SPLINE
SPL {X  -145.877, Y  +737.201, Z    +0.000, E1   +34.468, E3 -287162.055}
SPL {X  -152.550, Y  +719.721, Z    +0.000, E1   +27.728, E3 -287177.544}
SPL {X  -157.145, Y  +701.536, Z    +0.000, E1   +19.368, E3 -287186.999}
SPL {X  -159.035, Y  +688.952, Z    +0.000, E1   +12.676, E3 -287191.040}
SPL {X  -159.756, Y  +680.154, Z    +0.000, E1    +7.520, E3 -287192.766}
SPL {X  -159.986, Y  +672.560, Z    +0.000, E1    +2.636, E3 -287193.664}
SPL {X  -159.990, Y  +668.344, Z    +0.000, E1    -0.618, E3 -287193.931}
SPL {X  -159.990, Y  +664.070, Z    +0.000, E1    -5.025, E3 -287194.259}
SPL {X  -159.990, Y  +656.953, Z    +0.000, E1   -13.960, E3 -287195.325}
SPL {X  -159.990, Y  +644.589, Z    +0.000, E1   -29.011, E3 -287198.737}
SPL {X  -159.990, Y  +605.095, Z    +0.000, E1   -49.514, E3 -287223.828}
SPL {X  -159.990, Y  +543.998, Z    +0.000, E1   -54.483, E3 -287289.818}
SPL {X  -159.990, Y  +535.878, Z    +0.000, E1   -54.465, E3 -287302.152}
SPL {X  -159.990, Y  +529.394, Z    +0.000, E1   -54.464, E3 -287311.982}
SPL {X  -159.990, Y  +521.536, Z    +0.000, E1   -54.480, E3 -287323.864}
SPL {X  -159.990, Y  +512.119, Z    +0.000, E1   -54.487, E3 -287338.110}
SPL {X  -159.990, Y  +504.581, Z    +0.000, E1   -54.460, E3 -287349.569}
SPL {X  -159.990, Y  +497.571, Z    +0.000, E1   -54.478, E3 -287360.155}
SPL {X  -159.990, Y  +490.343, Z    +0.000, E1   -54.468, E3 -287371.121}
SPL {X  -159.990, Y  +483.191, Z    +0.000, E1   -54.478, E3 -287381.937}
SPL {X  -159.990, Y  +475.502, Z    +0.000, E1   -54.476, E3 -287393.586}
SPL {X  -159.990, Y  +448.520, Z    +0.000, E1   -58.543, E3 -287405.215}
SPL {X  -159.990, Y  +438.044, Z    +0.000, E1   -58.687, E3 -287417.852}
SPL {X  -159.990, Y  +431.936, Z    +0.000, E1   -57.955, E3 -287430.671}
SPL {X  -159.990, Y  +427.293, Z    +0.000, E1   -56.830, E3 -287444.377}
SPL {X  -159.990, Y  +423.841, Z    +0.000, E1   -55.679, E3 -287456.479}
SPL {X  -159.990, Y  +418.232, Z    +0.000, E1   -55.048, E3 -287468.833}
SPL {X  -159.990, Y  +410.722, Z    +0.000, E1   -54.900, E3 -287480.816}
SPL {X  -159.990, Y  +402.790, Z    +0.000, E1   -54.930, E3 -287492.591}
SPL {X  -159.990, Y  +392.953, Z    +0.000, E1   -54.918, E3 -287507.285}
SPL {X  -159.990, Y  +383.354, Z    +0.000, E1   -54.920, E3 -287521.595}
SPL {X  -159.769, Y  +374.091, Z    +0.000, E1   -54.882, E3 -287535.627}
SPL {X  -158.996, Y  +364.689, Z    +0.000, E1   -54.773, E3 -287550.424}
SPL {X  -157.966, Y  +357.131, Z    +0.000, E1   -54.559, E3 -287562.831}
SPL {X  -156.775, Y  +350.586, Z    +0.000, E1   -54.373, E3 -287573.805}
SPL {X  -155.027, Y  +342.959, Z    +0.000, E1   -54.074, E3 -287586.978}
SPL {X  -152.882, Y  +335.340, Z    +0.000, E1   -53.695, E3 -287600.520}
SPL {X  -151.019, Y  +329.680, Z    +0.000, E1   -53.334, E3 -287610.877}
SPL {X  -148.682, Y  +323.421, Z    +0.000, E1   -52.939, E3 -287622.480}
SPL {X  -145.914, Y  +316.881, Z    +0.000, E1   -52.402, E3 -287634.944}
SPL {X  -142.795, Y  +310.344, Z    +0.000, E1   -51.829, E3 -287647.600}
SPL {X  -132.354, Y  +292.616, Z    +0.000, E1   -44.164, E3 -287746.012}
ENDSPLINE

SPLINE
SPL {X  -150.910, Y  +329.369, Z    +0.000, E1   -29.678, E3 -287818.407}
SPL {X  -156.829, Y  +350.854, Z    +0.000, E1   -20.141, E3 -287830.960}
SPL {X  -159.049, Y  +365.169, Z    +0.000, E1   -12.580, E3 -287835.704}
SPL {X  -159.776, Y  +374.231, Z    +0.000, E1    -7.281, E3 -287837.590}
SPL {X  -159.986, Y  +381.380, Z    +0.000, E1    -2.685, E3 -287838.436}
SPL {X  -159.990, Y  +384.493, Z    +0.000, E1    -0.324, E3 -287838.644}
SPL {X  -159.990, Y  +387.327, Z    +0.000, E1    +2.137, E3 -287838.827}
SPL {X  -159.990, Y  +392.053, Z    +0.000, E1    +7.477, E3 -287839.292}
SPL {X  -159.990, Y  +396.158, Z    +0.000, E1   +12.775, E3 -287839.918}
SPL {X  -159.990, Y  +401.377, Z    +0.000, E1   +19.398, E3 -287841.098}
SPL {X  -159.990, Y  +411.365, Z    +0.000, E1   +30.630, E3 -287844.306}
SPL {X  -159.990, Y  +450.467, Z    +0.000, E1   +50.183, E3 -287867.955}
SPL {X  -159.990, Y  +509.934, Z    +0.000, E1   +54.923, E3 -287930.574}
SPL {X  -159.990, Y  +516.848, Z    +0.000, E1   +54.930, E3 -287940.862}
SPL {X  -159.990, Y  +524.818, Z    +0.000, E1   +54.933, E3 -287952.734}
SPL {X  -159.990, Y  +532.100, Z    +0.000, E1   +54.924, E3 -287963.587}
SPL {X  -159.990, Y  +539.391, Z    +0.000, E1   +54.933, E3 -287974.439}
SPL {X  -159.990, Y  +546.283, Z    +0.000, E1   +54.924, E3 -287984.711}
SPL {X  -159.990, Y  +553.734, Z    +0.000, E1   +54.938, E3 -287995.797}
SPL {X  -159.990, Y  +560.983, Z    +0.000, E1   +54.918, E3 -288006.635}
SPL {X  -159.990, Y  +567.462, Z    +0.000, E1   +54.929, E3 -288016.270}
SPL {X  -159.990, Y  +575.140, Z    +0.000, E1   +54.928, E3 -288027.702}
SPL {X  -159.990, Y  +581.046, Z    +0.000, E1   +54.920, E3 -288036.514}
SPL {X  -159.990, Y  +588.063, Z    +0.000, E1   +54.931, E3 -288046.949}
SPL {X  -159.990, Y  +595.273, Z    +0.000, E1   +54.928, E3 -288057.673}
SPL {X  -159.990, Y  +602.326, Z    +0.000, E1   +54.932, E3 -288068.173}
SPL {X  -159.990, Y  +610.296, Z    +0.000, E1   +54.937, E3 -288080.043}
SPL {X  -159.990, Y  +618.534, Z    +0.000, E1   +54.942, E3 -288092.280}
SPL {X  -159.990, Y  +628.178, Z    +0.000, E1   +54.959, E3 -288106.611}
SPL {X  -159.990, Y  +638.304, Z    +0.000, E1   +54.952, E3 -288121.700}
SPL {X  -159.990, Y  +645.976, Z    +0.000, E1   +54.934, E3 -288133.134}
SPL {X  -159.990, Y  +650.756, Z    +0.000, E1   +54.931, E3 -288140.249}
SPL {X  -159.990, Y  +658.525, Z    +0.000, E1   +54.959, E3 -288151.785}
SPL {X  -159.990, Y  +667.903, Z    +0.000, E1   +54.941, E3 -288165.816}
SPL {X  -159.827, Y  +678.718, Z    +0.000, E1   +54.950, E3 -288182.035}
SPL {X  -159.222, Y  +687.156, Z    +0.000, E1   +54.792, E3 -288195.346}
SPL {X  -158.388, Y  +694.082, Z    +0.000, E1   +54.679, E3 -288206.484}
SPL {X  -157.277, Y  +700.838, Z    +0.000, E1   +54.465, E3 -288217.741}
SPL {X  -156.153, Y  +706.327, Z    +0.000, E1   +54.274, E3 -288227.077}
SPL {X  -154.917, Y  +711.470, Z    +0.000, E1   +54.052, E3 -288236.029}
SPL {X  -153.204, Y  +717.603, Z    +0.000, E1   +53.775, E3 -288246.875}
SPL {X  -151.355, Y  +723.351, Z    +0.000, E1   +53.415, E3 -288257.346}
SPL {X  -149.371, Y  +728.816, Z    +0.000, E1   +53.074, E3 -288267.437}
SPL {X  -146.631, Y  +735.501, Z    +0.000, E1   +52.568, E3 -288280.097}
SPL {X  -144.428, Y  +740.329, Z    +0.000, E1   +52.109, E3 -288289.451}
SPL {X  -142.385, Y  +744.461, Z    +0.000, E1   +51.729, E3 -288297.502}
SPL {X  -132.301, Y  +761.463, Z    +0.000, E1   +45.510, E3 -288375.241}
ENDSPLINE

SPLINE
SPL {X  -145.877, Y  +737.201, Z    +0.000, E1   +34.468, E3 -288458.351}
SPL {X  -152.550, Y  +719.721, Z    +0.000, E1   +27.728, E3 -288473.841}
SPL {X  -157.145, Y  +701.536, Z    +0.000, E1   +19.368, E3 -288483.295}
SPL {X  -159.035, Y  +688.952, Z    +0.000, E1   +12.676, E3 -288487.336}
SPL {X  -159.756, Y  +680.154, Z    +0.000, E1    +7.520, E3 -288489.063}
SPL {X  -159.986, Y  +672.560, Z    +0.000, E1    +2.636, E3 -288489.961}
SPL {X  -159.990, Y  +668.344, Z    +0.000, E1    -0.618, E3 -288490.227}
SPL {X  -159.990, Y  +664.070, Z    +0.000, E1    -5.025, E3 -288490.555}
SPL {X  -159.990, Y  +656.953, Z    +0.000, E1   -13.960, E3 -288491.622}
SPL {X  -159.990, Y  +644.589, Z    +0.000, E1   -29.011, E3 -288495.033}
SPL {X  -159.990, Y  +605.095, Z    +0.000, E1   -49.514, E3 -288520.124}
SPL {X  -159.990, Y  +543.998, Z    +0.000, E1   -54.483, E3 -288586.114}
SPL {X  -159.990, Y  +535.878, Z    +0.000, E1   -54.465, E3 -288598.449}
SPL {X  -159.990, Y  +529.394, Z    +0.000, E1   -54.464, E3 -288608.278}
SPL {X  -159.990, Y  +521.536, Z    +0.000, E1   -54.480, E3 -288620.160}
SPL {X  -159.990, Y  +514.089, Z    +0.000, E1   -54.461, E3 -288631.472}
SPL {X  -159.990, Y  +506.373, Z    +0.000, E1   -54.484, E3 -288643.109}
SPL {X  -159.990, Y  +497.571, Z    +0.000, E1   -54.478, E3 -288656.452}
SPL {X  -159.990, Y  +490.343, Z    +0.000, E1   -54.468, E3 -288667.417}
SPL {X  -159.990, Y  +483.191, Z    +0.000, E1   -54.478, E3 -288678.233}
SPL {X  -159.990, Y  +475.502, Z    +0.000, E1   -54.476, E3 -288689.882}
SPL {X  -159.990, Y  +448.520, Z    +0.000, E1   -58.543, E3 -288701.511}
SPL {X  -159.990, Y  +438.044, Z    +0.000, E1   -58.687, E3 -288714.148}
SPL {X  -159.990, Y  +431.936, Z    +0.000, E1   -57.955, E3 -288726.968}
SPL {X  -159.990, Y  +427.860, Z    +0.000, E1   -57.091, E3 -288738.031}
SPL {X  -159.990, Y  +424.653, Z    +0.000, E1   -55.901, E3 -288750.337}
SPL {X  -159.990, Y  +419.589, Z    +0.000, E1   -55.096, E3 -288762.700}
SPL {X  -159.990, Y  +412.636, Z    +0.000, E1   -54.925, E3 -288774.212}
SPL {X  -159.990, Y  +405.235, Z    +0.000, E1   -54.902, E3 -288785.282}
SPL {X  -159.990, Y  +400.284, Z    +0.000, E1   -54.897, E3 -288792.677}
SPL {X  -159.990, Y  +392.953, Z    +0.000, E1   -54.918, E3 -288803.581}
SPL {X  -159.990, Y  +383.354, Z    +0.000, E1   -54.920, E3 -288817.891}
SPL {X  -159.860, Y  +376.053, Z    +0.000, E1   -54.872, E3 -288828.951}
SPL {X  -159.499, Y  +369.977, Z    +0.000, E1   -54.827, E3 -288838.356}
SPL {X  -158.803, Y  +363.045, Z    +0.000, E1   -54.709, E3 -288849.424}
SPL {X  -157.732, Y  +355.717, Z    +0.000, E1   -54.540, E3 -288861.447}
SPL {X  -156.235, Y  +348.039, Z    +0.000, E1   -54.281, E3 -288874.458}
SPL {X  -154.264, Y  +340.082, Z    +0.000, E1   -53.947, E3 -288888.335}
SPL {X  -151.643, Y  +331.497, Z    +0.000, E1   -53.493, E3 -288903.776}
SPL {X  -148.682, Y  +323.421, Z    +0.000, E1   -52.939, E3 -288918.776}
SPL {X  -145.914, Y  +316.881, Z    +0.000, E1   -52.402, E3 -288931.240}
SPL {X  -143.679, Y  +312.121, Z    +0.000, E1   -51.954, E3 -288940.485}
SPL {X  -141.812, Y  +308.430, Z    +0.000, E1   -51.590, E3 -288947.717}
SPL {X  -132.354, Y  +292.616, Z    +0.000, E1   -44.164, E3 -289042.308}
ENDSPLINE

SPLINE
SPL {X  -150.910, Y  +329.369, Z    +0.000, E1   -29.678, E3 -289114.704}
SPL {X  -156.829, Y  +350.854, Z    +0.000, E1   -20.141, E3 -289127.256}
SPL {X  -159.049, Y  +365.169, Z    +0.000, E1   -12.580, E3 -289132.000}
SPL {X  -159.776, Y  +374.231, Z    +0.000, E1    -7.281, E3 -289133.887}
SPL {X  -159.986, Y  +381.380, Z    +0.000, E1    -2.685, E3 -289134.733}
SPL {X  -159.990, Y  +384.493, Z    +0.000, E1    -0.324, E3 -289134.941}
SPL {X  -159.990, Y  +387.327, Z    +0.000, E1    +2.137, E3 -289135.123}
SPL {X  -159.990, Y  +392.053, Z    +0.000, E1    +7.477, E3 -289135.588}
SPL {X  -159.990, Y  +396.158, Z    +0.000, E1   +12.775, E3 -289136.214}
SPL {X  -159.990, Y  +401.377, Z    +0.000, E1   +19.398, E3 -289137.394}
SPL {X  -159.990, Y  +411.365, Z    +0.000, E1   +30.630, E3 -289140.603}
SPL {X  -159.990, Y  +450.467, Z    +0.000, E1   +50.183, E3 -289164.251}
SPL {X  -159.990, Y  +509.934, Z    +0.000, E1   +54.923, E3 -289226.870}
SPL {X  -159.990, Y  +516.848, Z    +0.000, E1   +54.930, E3 -289237.158}
SPL {X  -159.990, Y  +524.818, Z    +0.000, E1   +54.933, E3 -289249.030}
SPL {X  -159.990, Y  +532.100, Z    +0.000, E1   +54.924, E3 -289259.883}
SPL {X  -159.990, Y  +539.391, Z    +0.000, E1   +54.933, E3 -289270.735}
SPL {X  -159.990, Y  +546.283, Z    +0.000, E1   +54.924, E3 -289281.007}
SPL {X  -159.990, Y  +553.734, Z    +0.000, E1   +54.938, E3 -289292.094}
SPL {X  -159.990, Y  +564.956, Z    +0.000, E1   +54.973, E3 -289308.765}
SPL {X  -159.990, Y  +575.140, Z    +0.000, E1   +54.928, E3 -289323.998}
SPL {X  -159.990, Y  +581.046, Z    +0.000, E1   +54.920, E3 -289332.811}
SPL {X  -159.990, Y  +588.063, Z    +0.000, E1   +54.931, E3 -289343.246}
SPL {X  -159.990, Y  +595.273, Z    +0.000, E1   +54.928, E3 -289353.969}
SPL {X  -159.990, Y  +602.326, Z    +0.000, E1   +54.932, E3 -289364.470}
SPL {X  -159.990, Y  +610.296, Z    +0.000, E1   +54.937, E3 -289376.339}
SPL {X  -159.990, Y  +618.534, Z    +0.000, E1   +54.942, E3 -289388.576}
SPL {X  -159.990, Y  +625.928, Z    +0.000, E1   +54.931, E3 -289399.601}
SPL {X  -159.990, Y  +633.423, Z    +0.000, E1   +54.943, E3 -289410.743}
SPL {X  -159.990, Y  +640.333, Z    +0.000, E1   +54.927, E3 -289421.057}
SPL {X  -159.990, Y  +648.272, Z    +0.000, E1   +54.961, E3 -289432.805}
SPL {X  -159.990, Y  +655.990, Z    +0.000, E1   +54.930, E3 -289444.352}
SPL {X  -159.990, Y  +665.734, Z    +0.000, E1   +54.984, E3 -289458.804}
SPL {X  -159.953, Y  +674.920, Z    +0.000, E1   +54.918, E3 -289472.615}
SPL {X  -159.714, Y  +680.893, Z    +0.000, E1   +54.890, E3 -289481.755}
SPL {X  -159.222, Y  +687.156, Z    +0.000, E1   +54.792, E3 -289491.643}
SPL {X  -158.388, Y  +694.082, Z    +0.000, E1   +54.679, E3 -289502.780}
SPL {X  -157.277, Y  +700.838, Z    +0.000, E1   +54.465, E3 -289514.038}
SPL {X  -156.153, Y  +706.327, Z    +0.000, E1   +54.274, E3 -289523.374}
SPL {X  -154.505, Y  +713.032, Z    +0.000, E1   +54.006, E3 -289535.035}
SPL {X  -152.808, Y  +718.896, Z    +0.000, E1   +53.679, E3 -289545.532}
SPL {X  -150.773, Y  +725.019, Z    +0.000, E1   +53.343, E3 -289556.664}
SPL {X  -148.029, Y  +732.198, Z    +0.000, E1   +52.831, E3 -289570.101}
SPL {X  -145.158, Y  +738.775, Z    +0.000, E1   +52.288, E3 -289582.686}
SPL {X  -142.385, Y  +744.461, Z    +0.000, E1   +51.729, E3 -289593.798}
SPL {X  -132.301, Y  +761.463, Z    +0.000, E1   +45.510, E3 -289671.537}
ENDSPLINE

SPLINE
SPL {X  -145.877, Y  +737.201, Z    +0.000, E1   +34.468, E3 -289754.648}
SPL {X  -152.550, Y  +719.721, Z    +0.000, E1   +27.728, E3 -289770.137}
SPL {X  -157.145, Y  +701.536, Z    +0.000, E1   +19.368, E3 -289779.592}
SPL {X  -159.035, Y  +688.952, Z    +0.000, E1   +12.676, E3 -289783.633}
SPL {X  -159.756, Y  +680.154, Z    +0.000, E1    +7.520, E3 -289785.359}
SPL {X  -159.986, Y  +672.560, Z    +0.000, E1    +2.636, E3 -289786.257}
SPL {X  -159.990, Y  +668.344, Z    +0.000, E1    -0.618, E3 -289786.523}
SPL {X  -159.990, Y  +664.070, Z    +0.000, E1    -5.025, E3 -289786.852}
SPL {X  -159.990, Y  +656.953, Z    +0.000, E1   -13.960, E3 -289787.918}
SPL {X  -159.990, Y  +644.589, Z    +0.000, E1   -29.011, E3 -289791.330}
SPL {X  -159.990, Y  +605.095, Z    +0.000, E1   -49.514, E3 -289816.420}
SPL {X  -159.990, Y  +543.998, Z    +0.000, E1   -54.483, E3 -289882.410}
SPL {X  -159.990, Y  +535.878, Z    +0.000, E1   -54.465, E3 -289894.745}
SPL {X  -159.990, Y  +529.394, Z    +0.000, E1   -54.464, E3 -289904.575}
SPL {X  -159.990, Y  +521.536, Z    +0.000, E1   -54.480, E3 -289916.456}
SPL {X  -159.990, Y  +514.089, Z    +0.000, E1   -54.461, E3 -289927.769}
SPL {X  -159.990, Y  +506.373, Z    +0.000, E1   -54.484, E3 -289939.405}
SPL {X  -159.990, Y  +497.571, Z    +0.000, E1   -54.478, E3 -289952.748}
SPL {X  -159.990, Y  +490.343, Z    +0.000, E1   -54.468, E3 -289963.713}
SPL {X  -159.990, Y  +483.191, Z    +0.000, E1   -54.478, E3 -289974.529}
SPL {X  -159.990, Y  +471.543, Z    +0.000, E1   -55.096, E3 -289988.157}
SPL {X  -159.990, Y  +443.253, Z    +0.000, E1   -59.297, E3 -289999.589}
SPL {X  -159.990, Y  +438.044, Z    +0.000, E1   -58.687, E3 -290010.444}
SPL {X  -159.990, Y  +431.936, Z    +0.000, E1   -57.955, E3 -290023.264}
SPL {X  -159.990, Y  +427.860, Z    +0.000, E1   -57.091, E3 -290034.328}
SPL {X  -159.990, Y  +424.653, Z    +0.000, E1   -55.901, E3 -290046.633}
SPL {X  -159.990, Y  +418.232, Z    +0.000, E1   -55.048, E3 -290061.426}
SPL {X  -159.990, Y  +410.722, Z    +0.000, E1   -54.900, E3 -290073.409}
SPL {X  -159.990, Y  +402.790, Z    +0.000, E1   -54.930, E3 -290085.184}
SPL {X  -159.990, Y  +391.119, Z    +0.000, E1   -54.948, E3 -290102.561}
SPL {X  -159.951, Y  +378.972, Z    +0.000, E1   -54.929, E3 -290120.740}
SPL {X  -159.499, Y  +369.977, Z    +0.000, E1   -54.827, E3 -290134.652}
SPL {X  -158.803, Y  +363.045, Z    +0.000, E1   -54.709, E3 -290145.721}
SPL {X  -157.966, Y  +357.131, Z    +0.000, E1   -54.559, E3 -290155.424}
SPL {X  -156.775, Y  +350.586, Z    +0.000, E1   -54.373, E3 -290166.397}
SPL {X  -155.027, Y  +342.959, Z    +0.000, E1   -54.074, E3 -290179.570}
SPL {X  -152.882, Y  +335.340, Z    +0.000, E1   -53.695, E3 -290193.113}
SPL {X  -151.019, Y  +329.680, Z    +0.000, E1   -53.334, E3 -290203.470}
SPL {X  -149.351, Y  +325.131, Z    +0.000, E1   -53.025, E3 -290211.914}
SPL {X  -147.860, Y  +321.391, Z    +0.000, E1   -52.740, E3 -290218.967}
SPL {X  -145.914, Y  +316.881, Z    +0.000, E1   -52.402, E3 -290227.536}
SPL {X  -142.795, Y  +310.344, Z    +0.000, E1   -51.829, E3 -290240.192}
SPL {X  -132.354, Y  +292.616, Z    +0.000, E1   -44.164, E3 -290338.604}
ENDSPLINE

SPLINE
SPL {X  -150.910, Y  +329.369, Z    +0.000, E1   -29.678, E3 -290411.000}
SPL {X  -156.396, Y  +348.778, Z    +0.000, E1   -21.134, E3 -290422.643}
SPL {X  -158.554, Y  +361.116, Z    +0.000, E1   -14.883, E3 -290427.097}
SPL {X  -159.881, Y  +376.607, Z    +0.000, E1    -5.865, E3 -290430.506}
SPL {X  -159.990, Y  +383.659, Z    +0.000, E1    -1.050, E3 -290431.187}
SPL {X  -159.990, Y  +387.327, Z    +0.000, E1    +2.137, E3 -290431.420}
SPL {X  -159.990, Y  +390.622, Z    +0.000, E1    +5.876, E3 -290431.713}
SPL {X  -159.990, Y  +394.493, Z    +0.000, E1   +10.512, E3 -290432.236}
SPL {X  -159.990, Y  +401.377, Z    +0.000, E1   +19.398, E3 -290433.690}
SPL {X  -159.990, Y  +411.365, Z    +0.000, E1   +30.630, E3 -290436.899}
SPL {X  -159.990, Y  +450.467, Z    +0.000, E1   +50.183, E3 -290460.548}
SPL {X  -159.990, Y  +509.934, Z    +0.000, E1   +54.923, E3 -290523.167}
SPL {X  -159.990, Y  +516.848, Z    +0.000, E1   +54.930, E3 -290533.455}
SPL {X  -159.990, Y  +524.818, Z    +0.000, E1   +54.933, E3 -290545.327}
SPL {X  -159.990, Y  +532.100, Z    +0.000, E1   +54.924, E3 -290556.180}
SPL {X  -159.990, Y  +539.391, Z    +0.000, E1   +54.933, E3 -290567.032}
SPL {X  -159.990, Y  +546.283, Z    +0.000, E1   +54.924, E3 -290577.303}
SPL {X  -159.990, Y  +553.734, Z    +0.000, E1   +54.938, E3 -290588.390}
SPL {X  -159.990, Y  +564.956, Z    +0.000, E1   +54.973, E3 -290605.061}
SPL {X  -159.990, Y  +577.902, Z    +0.000, E1   +54.969, E3 -290624.351}
SPL {X  -159.990, Y  +588.063, Z    +0.000, E1   +54.931, E3 -290639.542}
SPL {X  -159.990, Y  +595.273, Z    +0.000, E1   +54.928, E3 -290650.265}
SPL {X  -159.990, Y  +602.326, Z    +0.000, E1   +54.932, E3 -290660.766}
SPL {X  -159.990, Y  +610.296, Z    +0.000, E1   +54.937, E3 -290672.635}
SPL {X  -159.990, Y  +618.534, Z    +0.000, E1   +54.942, E3 -290684.872}
SPL {X  -159.990, Y  +628.178, Z    +0.000, E1   +54.959, E3 -290699.203}
SPL {X  -159.990, Y  +638.304, Z    +0.000, E1   +54.952, E3 -290714.292}
SPL {X  -159.990, Y  +648.272, Z    +0.000, E1   +54.961, E3 -290729.101}
SPL {X  -159.990, Y  +655.990, Z    +0.000, E1   +54.930, E3 -290740.649}
SPL {X  -159.990, Y  +665.734, Z    +0.000, E1   +54.984, E3 -290755.100}
SPL {X  -159.827, Y  +678.718, Z    +0.000, E1   +54.950, E3 -290774.628}
SPL {X  -159.222, Y  +687.156, Z    +0.000, E1   +54.792, E3 -290787.939}
SPL {X  -158.388, Y  +694.082, Z    +0.000, E1   +54.679, E3 -290799.077}
SPL {X  -157.277, Y  +700.838, Z    +0.000, E1   +54.465, E3 -290810.334}
SPL {X  -156.153, Y  +706.327, Z    +0.000, E1   +54.274, E3 -290819.670}
SPL {X  -154.917, Y  +711.470, Z    +0.000, E1   +54.052, E3 -290828.621}
SPL {X  -153.204, Y  +717.603, Z    +0.000, E1   +53.775, E3 -290839.467}
SPL {X  -151.355, Y  +723.351, Z    +0.000, E1   +53.415, E3 -290849.939}
SPL {X  -149.371, Y  +728.816, Z    +0.000, E1   +53.074, E3 -290860.029}
SPL {X  -147.376, Y  +733.767, Z    +0.000, E1   +52.671, E3 -290869.431}
SPL {X  -145.158, Y  +738.775, Z    +0.000, E1   +52.288, E3 -290878.982}
SPL {X  -142.385, Y  +744.461, Z    +0.000, E1   +51.729, E3 -290890.094}
SPL {X  -132.301, Y  +761.463, Z    +0.000, E1   +45.510, E3 -290967.833}
ENDSPLINE

SPLINE
SPL {X  -145.877, Y  +737.201, Z    +0.000, E1   +34.468, E3 -291050.944}
SPL {X  -152.550, Y  +719.721, Z    +0.000, E1   +27.728, E3 -291066.433}
SPL {X  -157.145, Y  +701.536, Z    +0.000, E1   +19.368, E3 -291075.888}
SPL {X  -159.035, Y  +688.952, Z    +0.000, E1   +12.676, E3 -291079.929}
SPL {X  -159.756, Y  +680.154, Z    +0.000, E1    +7.520, E3 -291081.655}
SPL {X  -159.986, Y  +672.560, Z    +0.000, E1    +2.636, E3 -291082.553}
SPL {X  -159.990, Y  +668.344, Z    +0.000, E1    -0.618, E3 -291082.819}
SPL {X  -159.990, Y  +664.070, Z    +0.000, E1    -5.025, E3 -291083.148}
SPL {X  -159.990, Y  +656.953, Z    +0.000, E1   -13.960, E3 -291084.214}
SPL {X  -159.990, Y  +644.589, Z    +0.000, E1   -29.011, E3 -291087.626}
SPL {X  -159.990, Y  +605.095, Z    +0.000, E1   -49.514, E3 -291112.717}
SPL {X  -159.990, Y  +546.155, Z    +0.000, E1   -54.461, E3 -291175.475}
SPL {X  -159.990, Y  +537.700, Z    +0.000, E1   -54.492, E3 -291188.239}
SPL {X  -159.990, Y  +529.394, Z    +0.000, E1   -54.464, E3 -291200.871}
SPL {X  -159.990, Y  +521.536, Z    +0.000, E1   -54.480, E3 -291212.753}
SPL {X  -159.990, Y  +514.089, Z    +0.000, E1   -54.461, E3 -291224.065}
SPL {X  -159.990, Y  +506.373, Z    +0.000, E1   -54.484, E3 -291235.701}
SPL {X  -159.990, Y  +497.571, Z    +0.000, E1   -54.478, E3 -291249.044}
SPL {X  -159.990, Y  +490.343, Z    +0.000, E1   -54.468, E3 -291260.009}
SPL {X  -159.990, Y  +483.191, Z    +0.000, E1   -54.478, E3 -291270.826}
SPL {X  -159.990, Y  +475.502, Z    +0.000, E1   -54.476, E3 -291282.475}
SPL {X  -159.990, Y  +448.520, Z    +0.000, E1   -58.543, E3 -291294.104}
SPL {X  -159.990, Y  +438.044, Z    +0.000, E1   -58.687, E3 -291306.741}
SPL {X  -159.990, Y  +431.936, Z    +0.000, E1   -57.955, E3 -291319.560}
SPL {X  -159.990, Y  +427.860, Z    +0.000, E1   -57.091, E3 -291330.624}
SPL {X  -159.990, Y  +424.653, Z    +0.000, E1   -55.901, E3 -291342.929}
SPL {X  -159.990, Y  +418.232, Z    +0.000, E1   -55.048, E3 -291357.722}
SPL {X  -159.990, Y  +410.722, Z    +0.000, E1   -54.900, E3 -291369.705}
SPL {X  -159.990, Y  +402.790, Z    +0.000, E1   -54.930, E3 -291381.480}
SPL {X  -159.990, Y  +392.953, Z    +0.000, E1   -54.918, E3 -291396.174}
SPL {X  -159.990, Y  +383.354, Z    +0.000, E1   -54.920, E3 -291410.484}
SPL {X  -159.860, Y  +376.053, Z    +0.000, E1   -54.872, E3 -291421.544}
SPL {X  -159.499, Y  +369.977, Z    +0.000, E1   -54.827, E3 -291430.948}
SPL {X  -158.803, Y  +363.045, Z    +0.000, E1   -54.709, E3 -291442.017}
SPL {X  -157.732, Y  +355.717, Z    +0.000, E1   -54.540, E3 -291454.039}
SPL {X  -156.235, Y  +348.039, Z    +0.000, E1   -54.281, E3 -291467.051}
SPL {X  -154.716, Y  +341.761, Z    +0.000, E1   -53.995, E3 -291478.008}
SPL {X  -152.882, Y  +335.340, Z    +0.000, E1   -53.695, E3 -291489.409}
SPL {X  -151.019, Y  +329.680, Z    +0.000, E1   -53.334, E3 -291499.766}
SPL {X  -149.351, Y  +325.131, Z    +0.000, E1   -53.025, E3 -291508.210}
SPL {X  -147.860, Y  +321.391, Z    +0.000, E1   -52.740, E3 -291515.263}
SPL {X  -145.914, Y  +316.881, Z    +0.000, E1   -52.402, E3 -291523.833}
SPL {X  -142.795, Y  +310.344, Z    +0.000, E1   -51.829, E3 -291536.488}
SPL {X  -132.354, Y  +292.616, Z    +0.000, E1   -44.164, E3 -291634.901}
ENDSPLINE

SPLINE
SPL {X  -150.910, Y  +329.369, Z    +0.000, E1   -29.678, E3 -291707.296}
SPL {X  -156.829, Y  +350.854, Z    +0.000, E1   -20.141, E3 -291719.849}
SPL {X  -159.049, Y  +365.169, Z    +0.000, E1   -12.580, E3 -291724.593}
SPL {X  -159.776, Y  +374.231, Z    +0.000, E1    -7.281, E3 -291726.479}
SPL {X  -159.986, Y  +381.380, Z    +0.000, E1    -2.685, E3 -291727.325}
SPL {X  -159.990, Y  +384.493, Z    +0.000, E1    -0.324, E3 -291727.533}
SPL {X  -159.990, Y  +387.327, Z    +0.000, E1    +2.137, E3 -291727.716}
SPL {X  -159.990, Y  +392.053, Z    +0.000, E1    +7.477, E3 -291728.181}
SPL {X  -159.990, Y  +396.158, Z    +0.000, E1   +12.775, E3 -291728.806}
SPL {X  -159.990, Y  +401.377, Z    +0.000, E1   +19.398, E3 -291729.987}
SPL {X  -159.990, Y  +411.365, Z    +0.000, E1   +30.630, E3 -291733.195}
SPL {X  -159.990, Y  +450.467, Z    +0.000, E1   +50.183, E3 -291756.844}
SPL {X  -159.990, Y  +509.934, Z    +0.000, E1   +54.923, E3 -291819.463}
SPL {X  -159.990, Y  +516.848, Z    +0.000, E1   +54.930, E3 -291829.751}
SPL {X  -159.990, Y  +524.818, Z    +0.000, E1   +54.933, E3 -291841.623}
SPL {X  -159.990, Y  +532.100, Z    +0.000, E1   +54.924, E3 -291852.476}
SPL {X  -159.990, Y  +539.391, Z    +0.000, E1   +54.933, E3 -291863.328}
SPL {X  -159.990, Y  +546.283, Z    +0.000, E1   +54.924, E3 -291873.600}
SPL {X  -159.990, Y  +553.734, Z    +0.000, E1   +54.938, E3 -291884.686}
SPL {X  -159.990, Y  +560.983, Z    +0.000, E1   +54.918, E3 -291895.524}
SPL {X  -159.990, Y  +567.462, Z    +0.000, E1   +54.929, E3 -291905.159}
SPL {X  -159.990, Y  +575.140, Z    +0.000, E1   +54.928, E3 -291916.591}
SPL {X  -159.990, Y  +581.046, Z    +0.000, E1   +54.920, E3 -291925.403}
SPL {X  -159.990, Y  +588.063, Z    +0.000, E1   +54.931, E3 -291935.838}
SPL {X  -159.990, Y  +595.273, Z    +0.000, E1   +54.928, E3 -291946.562}
SPL {X  -159.990, Y  +602.326, Z    +0.000, E1   +54.932, E3 -291957.062}
SPL {X  -159.990, Y  +610.296, Z    +0.000, E1   +54.937, E3 -291968.932}
SPL {X  -159.990, Y  +618.534, Z    +0.000, E1   +54.942, E3 -291981.169}
SPL {X  -159.990, Y  +625.928, Z    +0.000, E1   +54.931, E3 -291992.194}
SPL {X  -159.990, Y  +633.423, Z    +0.000, E1   +54.943, E3 -292003.336}
SPL {X  -159.990, Y  +643.352, Z    +0.000, E1   +54.966, E3 -292018.071}
SPL {X  -159.990, Y  +650.756, Z    +0.000, E1   +54.931, E3 -292029.138}
SPL {X  -159.990, Y  +658.525, Z    +0.000, E1   +54.959, E3 -292040.674}
SPL {X  -159.990, Y  +667.903, Z    +0.000, E1   +54.941, E3 -292054.705}
SPL {X  -159.953, Y  +674.920, Z    +0.000, E1   +54.918, E3 -292065.208}
SPL {X  -159.714, Y  +680.893, Z    +0.000, E1   +54.890, E3 -292074.348}
SPL {X  -159.222, Y  +687.156, Z    +0.000, E1   +54.792, E3 -292084.235}
SPL {X  -158.388, Y  +694.082, Z    +0.000, E1   +54.679, E3 -292095.373}
SPL {X  -157.277, Y  +700.838, Z    +0.000, E1   +54.465, E3 -292106.630}
SPL {X  -156.153, Y  +706.327, Z    +0.000, E1   +54.274, E3 -292115.966}
SPL {X  -154.917, Y  +711.470, Z    +0.000, E1   +54.052, E3 -292124.917}
SPL {X  -153.204, Y  +717.603, Z    +0.000, E1   +53.775, E3 -292135.763}
SPL {X  -151.355, Y  +723.351, Z    +0.000, E1   +53.415, E3 -292146.235}
SPL {X  -149.371, Y  +728.816, Z    +0.000, E1   +53.074, E3 -292156.326}
SPL {X  -146.631, Y  +735.501, Z    +0.000, E1   +52.568, E3 -292168.986}
SPL {X  -144.428, Y  +740.329, Z    +0.000, E1   +52.109, E3 -292178.340}
SPL {X  -142.385, Y  +744.461, Z    +0.000, E1   +51.729, E3 -292186.391}
SPL {X  -132.301, Y  +761.463, Z    +0.000, E1   +45.510, E3 -292264.129}
ENDSPLINE

SPLINE
SPL {X  -145.877, Y  +737.201, Z    +0.000, E1   +34.468, E3 -292347.240}
SPL {X  -152.550, Y  +719.721, Z    +0.000, E1   +27.728, E3 -292362.729}
SPL {X  -157.145, Y  +701.536, Z    +0.000, E1   +19.368, E3 -292372.184}
SPL {X  -159.035, Y  +688.952, Z    +0.000, E1   +12.676, E3 -292376.225}
SPL {X  -159.756, Y  +680.154, Z    +0.000, E1    +7.520, E3 -292377.952}
SPL {X  -159.986, Y  +672.560, Z    +0.000, E1    +2.636, E3 -292378.850}
SPL {X  -159.990, Y  +668.344, Z    +0.000, E1    -0.618, E3 -292379.116}
SPL {X  -159.990, Y  +665.430, Z    +0.000, E1    -3.630, E3 -292379.311}
SPL {X  -159.990, Y  +661.750, Z    +0.000, E1    -7.880, E3 -292379.702}
SPL {X  -159.990, Y  +657.656, Z    +0.000, E1   -13.276, E3 -292380.347}
SPL {X  -159.990, Y  +652.023, Z    +0.000, E1   -20.449, E3 -292381.635}
SPL {X  -159.990, Y  +641.935, Z    +0.000, E1   -31.848, E3 -292384.807}
SPL {X  -159.990, Y  +605.095, Z    +0.000, E1   -49.514, E3 -292409.013}
SPL {X  -159.990, Y  +546.155, Z    +0.000, E1   -54.461, E3 -292471.772}
SPL {X  -159.990, Y  +537.700, Z    +0.000, E1   -54.492, E3 -292484.535}
SPL {X  -159.990, Y  +529.394, Z    +0.000, E1   -54.464, E3 -292497.167}
SPL {X  -159.990, Y  +521.536, Z    +0.000, E1   -54.480, E3 -292509.049}
SPL {X  -159.990, Y  +512.119, Z    +0.000, E1   -54.487, E3 -292523.295}
SPL {X  -159.990, Y  +504.581, Z    +0.000, E1   -54.460, E3 -292534.754}
SPL {X  -159.990, Y  +497.571, Z    +0.000, E1   -54.478, E3 -292545.341}
SPL {X  -159.990, Y  +490.343, Z    +0.000, E1   -54.468, E3 -292556.306}
SPL {X  -159.990, Y  +483.191, Z    +0.000, E1   -54.478, E3 -292567.122}
SPL {X  -159.990, Y  +475.502, Z    +0.000, E1   -54.476, E3 -292578.771}
SPL {X  -159.990, Y  +448.520, Z    +0.000, E1   -58.543, E3 -292590.400}
SPL {X  -159.990, Y  +438.044, Z    +0.000, E1   -58.687, E3 -292603.037}
SPL {X  -159.990, Y  +431.936, Z    +0.000, E1   -57.955, E3 -292615.857}
SPL {X  -159.990, Y  +427.293, Z    +0.000, E1   -56.830, E3 -292629.563}
SPL {X  -159.990, Y  +423.841, Z    +0.000, E1   -55.679, E3 -292641.664}
SPL {X  -159.990, Y  +418.232, Z    +0.000, E1   -55.048, E3 -292654.018}
SPL {X  -159.990, Y  +410.722, Z    +0.000, E1   -54.900, E3 -292666.001}
SPL {X  -159.990, Y  +402.790, Z    +0.000, E1   -54.930, E3 -292677.776}
SPL {X  -159.990, Y  +391.119, Z    +0.000, E1   -54.948, E3 -292695.154}
SPL {X  -159.951, Y  +378.972, Z    +0.000, E1   -54.929, E3 -292713.332}
SPL {X  -159.499, Y  +369.977, Z    +0.000, E1   -54.827, E3 -292727.245}
SPL {X  -158.803, Y  +363.045, Z    +0.000, E1   -54.709, E3 -292738.313}
SPL {X  -157.966, Y  +357.131, Z    +0.000, E1   -54.559, E3 -292748.016}
SPL {X  -156.775, Y  +350.586, Z    +0.000, E1   -54.373, E3 -292758.990}
SPL {X  -155.027, Y  +342.959, Z    +0.000, E1   -54.074, E3 -292772.163}
SPL {X  -153.580, Y  +337.668, Z    +0.000, E1   -53.781, E3 -292781.586}
SPL {X  -151.643, Y  +331.497, Z    +0.000, E1   -53.493, E3 -292792.665}
SPL {X  -148.682, Y  +323.421, Z    +0.000, E1   -52.939, E3 -292807.665}
SPL {X  -145.914, Y  +316.881, Z    +0.000, E1   -52.402, E3 -292820.129}
SPL {X  -142.795, Y  +310.344, Z    +0.000, E1   -51.829, E3 -292832.785}
SPL {X  -132.354, Y  +292.616, Z    +0.000, E1   -44.164, E3 -292931.197}
ENDSPLINE

SPLINE
SPL {X  -150.910, Y  +329.369, Z    +0.000, E1   -29.678, E3 -293003.593}
SPL {X  -156.829, Y  +350.854, Z    +0.000, E1   -20.141, E3 -293016.145}
SPL {X  -159.049, Y  +365.169, Z    +0.000, E1   -12.580, E3 -293020.889}
SPL {X  -159.776, Y  +374.231, Z    +0.000, E1    -7.281, E3 -293022.775}
SPL {X  -159.986, Y  +381.380, Z    +0.000, E1    -2.685, E3 -293023.621}
SPL {X  -159.990, Y  +385.261, Z    +0.000, E1    +0.259, E3 -293023.875}
SPL {X  -159.990, Y  +388.094, Z    +0.000, E1    +3.012, E3 -293024.067}
SPL {X  -159.990, Y  +390.622, Z    +0.000, E1    +5.876, E3 -293024.306}
SPL {X  -159.990, Y  +394.493, Z    +0.000, E1   +10.512, E3 -293024.829}
SPL {X  -159.990, Y  +401.377, Z    +0.000, E1   +19.398, E3 -293026.283}
SPL {X  -159.990, Y  +411.365, Z    +0.000, E1   +30.630, E3 -293029.491}
SPL {X  -159.990, Y  +450.467, Z    +0.000, E1   +50.183, E3 -293053.140}
SPL {X  -159.990, Y  +509.934, Z    +0.000, E1   +54.923, E3 -293115.759}
SPL {X  -159.990, Y  +516.848, Z    +0.000, E1   +54.930, E3 -293126.047}
SPL {X  -159.990, Y  +524.818, Z    +0.000, E1   +54.933, E3 -293137.919}
SPL {X  -159.990, Y  +532.100, Z    +0.000, E1   +54.924, E3 -293148.772}
SPL {X  -159.990, Y  +539.391, Z    +0.000, E1   +54.933, E3 -293159.624}
SPL {X  -159.990, Y  +546.283, Z    +0.000, E1   +54.924, E3 -293169.896}
SPL {X  -159.990, Y  +553.734, Z    +0.000, E1   +54.938, E3 -293180.983}
SPL {X  -159.990, Y  +564.956, Z    +0.000, E1   +54.973, E3 -293197.654}
SPL {X  -159.990, Y  +577.902, Z    +0.000, E1   +54.969, E3 -293216.944}
SPL {X  -159.990, Y  +588.063, Z    +0.000, E1   +54.931, E3 -293232.134}
SPL {X  -159.990, Y  +595.273, Z    +0.000, E1   +54.928, E3 -293242.858}
SPL {X  -159.990, Y  +602.326, Z    +0.000, E1   +54.932, E3 -293253.358}
SPL {X  -159.990, Y  +610.296, Z    +0.000, E1   +54.937, E3 -293265.228}
SPL {X  -159.990, Y  +618.534, Z    +0.000, E1   +54.942, E3 -293277.465}
SPL {X  -159.990, Y  +625.928, Z    +0.000, E1   +54.931, E3 -293288.490}
SPL {X  -159.990, Y  +633.423, Z    +0.000, E1   +54.943, E3 -293299.632}
SPL {X  -159.990, Y  +640.333, Z    +0.000, E1   +54.927, E3 -293309.946}
SPL {X  -159.990, Y  +648.272, Z    +0.000, E1   +54.961, E3 -293321.694}
SPL {X  -159.990, Y  +655.990, Z    +0.000, E1   +54.930, E3 -293333.241}
SPL {X  -159.990, Y  +665.734, Z    +0.000, E1   +54.984, E3 -293347.692}
SPL {X  -159.827, Y  +678.718, Z    +0.000, E1   +54.950, E3 -293367.221}
SPL {X  -159.222, Y  +687.156, Z    +0.000, E1   +54.792, E3 -293380.532}
SPL {X  -158.388, Y  +694.082, Z    +0.000, E1   +54.679, E3 -293391.669}
SPL {X  -157.277, Y  +700.838, Z    +0.000, E1   +54.465, E3 -293402.926}
SPL {X  -156.153, Y  +706.327, Z    +0.000, E1   +54.274, E3 -293412.262}
SPL {X  -154.917, Y  +711.470, Z    +0.000, E1   +54.052, E3 -293421.214}
SPL {X  -153.204, Y  +717.603, Z    +0.000, E1   +53.775, E3 -293432.060}
SPL {X  -151.355, Y  +723.351, Z    +0.000, E1   +53.415, E3 -293442.531}
SPL {X  -149.371, Y  +728.816, Z    +0.000, E1   +53.074, E3 -293452.622}
SPL {X  -147.376, Y  +733.767, Z    +0.000, E1   +52.671, E3 -293462.024}
SPL {X  -145.158, Y  +738.775, Z    +0.000, E1   +52.288, E3 -293471.575}
SPL {X  -142.385, Y  +744.461, Z    +0.000, E1   +51.729, E3 -293482.687}
SPL {X  -132.301, Y  +761.463, Z    +0.000, E1   +45.510, E3 -293560.426}
ENDSPLINE

SPLINE
SPL {X  -145.877, Y  +737.201, Z    +0.000, E1   +34.468, E3 -293643.537}
SPL {X  -152.550, Y  +719.721, Z    +0.000, E1   +27.728, E3 -293659.026}
SPL {X  -157.145, Y  +701.536, Z    +0.000, E1   +19.368, E3 -293668.480}
SPL {X  -159.035, Y  +688.952, Z    +0.000, E1   +12.676, E3 -293672.521}
SPL {X  -159.756, Y  +680.154, Z    +0.000, E1    +7.520, E3 -293674.248}
SPL {X  -159.986, Y  +672.560, Z    +0.000, E1    +2.636, E3 -293675.146}
SPL {X  -159.990, Y  +668.344, Z    +0.000, E1    -0.618, E3 -293675.412}
SPL {X  -159.990, Y  +664.070, Z    +0.000, E1    -5.025, E3 -293675.740}
SPL {X  -159.990, Y  +656.953, Z    +0.000, E1   -13.960, E3 -293676.807}
SPL {X  -159.990, Y  +644.589, Z    +0.000, E1   -29.011, E3 -293680.218}
SPL {X  -159.990, Y  +605.095, Z    +0.000, E1   -49.514, E3 -293705.309}
SPL {X  -159.990, Y  +543.998, Z    +0.000, E1   -54.483, E3 -293771.299}
SPL {X  -159.990, Y  +535.878, Z    +0.000, E1   -54.465, E3 -293783.634}
SPL {X  -159.990, Y  +529.394, Z    +0.000, E1   -54.464, E3 -293793.463}
SPL {X  -159.990, Y  +521.536, Z    +0.000, E1   -54.480, E3 -293805.345}
SPL {X  -159.990, Y  +514.089, Z    +0.000, E1   -54.461, E3 -293816.658}
SPL {X  -159.990, Y  +506.373, Z    +0.000, E1   -54.484, E3 -293828.294}
SPL {X  -159.990, Y  +497.571, Z    +0.000, E1   -54.478, E3 -293841.637}
SPL {X  -159.990, Y  +490.343, Z    +0.000, E1   -54.468, E3 -293852.602}
SPL {X  -159.990, Y  +483.191, Z    +0.000, E1   -54.478, E3 -293863.418}
SPL {X  -159.990, Y  +471.543, Z    +0.000, E1   -55.096, E3 -293877.046}
SPL {X  -159.990, Y  +443.253, Z    +0.000, E1   -59.297, E3 -293888.478}
SPL {X  -159.990, Y  +438.044, Z    +0.000, E1   -58.687, E3 -293899.333}
SPL {X  -159.990, Y  +431.936, Z    +0.000, E1   -57.955, E3 -293912.153}
SPL {X  -159.990, Y  +427.860, Z    +0.000, E1   -57.091, E3 -293923.216}
SPL {X  -159.990, Y  +424.653, Z    +0.000, E1   -55.901, E3 -293935.522}
SPL {X  -159.990, Y  +418.232, Z    +0.000, E1   -55.048, E3 -293950.315}
SPL {X  -159.990, Y  +410.722, Z    +0.000, E1   -54.900, E3 -293962.298}
SPL {X  -159.990, Y  +402.790, Z    +0.000, E1   -54.930, E3 -293974.073}
SPL {X  -159.990, Y  +391.119, Z    +0.000, E1   -54.948, E3 -293991.450}
SPL {X  -159.951, Y  +378.972, Z    +0.000, E1   -54.929, E3 -294009.629}
SPL {X  -159.499, Y  +369.977, Z    +0.000, E1   -54.827, E3 -294023.541}
SPL {X  -158.803, Y  +363.045, Z    +0.000, E1   -54.709, E3 -294034.609}
SPL {X  -157.966, Y  +357.131, Z    +0.000, E1   -54.559, E3 -294044.312}
SPL {X  -156.775, Y  +350.586, Z    +0.000, E1   -54.373, E3 -294055.286}
SPL {X  -155.027, Y  +342.959, Z    +0.000, E1   -54.074, E3 -294068.459}
SPL {X  -152.882, Y  +335.340, Z    +0.000, E1   -53.695, E3 -294082.002}
SPL {X  -151.019, Y  +329.680, Z    +0.000, E1   -53.334, E3 -294092.359}
SPL {X  -149.351, Y  +325.131, Z    +0.000, E1   -53.025, E3 -294100.803}
SPL {X  -147.860, Y  +321.391, Z    +0.000, E1   -52.740, E3 -294107.856}
SPL {X  -145.914, Y  +316.881, Z    +0.000, E1   -52.402, E3 -294116.425}
SPL {X  -142.795, Y  +310.344, Z    +0.000, E1   -51.829, E3 -294129.081}
SPL {X  -132.354, Y  +292.616, Z    +0.000, E1   -44.164, E3 -294227.493}
ENDSPLINE

SPLINE
SPL {X  -150.910, Y  +329.369, Z    +0.000, E1   -29.678, E3 -294299.889}
SPL {X  -156.396, Y  +348.778, Z    +0.000, E1   -21.134, E3 -294311.532}
SPL {X  -158.554, Y  +361.116, Z    +0.000, E1   -14.883, E3 -294315.986}
SPL {X  -159.881, Y  +376.607, Z    +0.000, E1    -5.865, E3 -294319.395}
SPL {X  -159.990, Y  +383.659, Z    +0.000, E1    -1.050, E3 -294320.076}
SPL {X  -159.990, Y  +387.327, Z    +0.000, E1    +2.137, E3 -294320.309}
SPL {X  -159.990, Y  +390.622, Z    +0.000, E1    +5.876, E3 -294320.602}
SPL {X  -159.990, Y  +394.493, Z    +0.000, E1   +10.512, E3 -294321.125}
SPL {X  -159.990, Y  +401.377, Z    +0.000, E1   +19.398, E3 -294322.579}
SPL {X  -159.990, Y  +411.365, Z    +0.000, E1   +30.630, E3 -294325.788}
SPL {X  -159.990, Y  +450.467, Z    +0.000, E1   +50.183, E3 -294349.437}
SPL {X  -159.990, Y  +509.934, Z    +0.000, E1   +54.923, E3 -294412.055}
SPL {X  -159.990, Y  +516.848, Z    +0.000, E1   +54.930, E3 -294422.344}
SPL {X  -159.990, Y  +524.818, Z    +0.000, E1   +54.933, E3 -294434.215}
SPL {X  -159.990, Y  +532.100, Z    +0.000, E1   +54.924, E3 -294445.068}
SPL {X  -159.990, Y  +539.391, Z    +0.000, E1   +54.933, E3 -294455.920}
SPL {X  -159.990, Y  +546.283, Z    +0.000, E1   +54.924, E3 -294466.192}
SPL {X  -159.990, Y  +553.734, Z    +0.000, E1   +54.938, E3 -294477.279}
SPL {X  -159.990, Y  +564.956, Z    +0.000, E1   +54.973, E3 -294493.950}
SPL {X  -159.990, Y  +577.902, Z    +0.000, E1   +54.969, E3 -294513.240}
SPL {X  -159.990, Y  +588.063, Z    +0.000, E1   +54.931, E3 -294528.431}
SPL {X  -159.990, Y  +595.273, Z    +0.000, E1   +54.928, E3 -294539.154}
SPL {X  -159.990, Y  +602.326, Z    +0.000, E1   +54.932, E3 -294549.655}
SPL {X  -159.990, Y  +610.296, Z    +0.000, E1   +54.937, E3 -294561.524}
SPL {X  -159.990, Y  +618.534, Z    +0.000, E1   +54.942, E3 -294573.761}
SPL {X  -159.990, Y  +628.178, Z    +0.000, E1   +54.959, E3 -294588.092}
SPL {X  -159.990, Y  +638.304, Z    +0.000, E1   +54.952, E3 -294603.181}
SPL {X  -159.990, Y  +648.272, Z    +0.000, E1   +54.961, E3 -294617.990}
SPL {X  -159.990, Y  +655.990, Z    +0.000, E1   +54.930, E3 -294629.538}
SPL {X  -159.990, Y  +665.734, Z    +0.000, E1   +54.984, E3 -294643.989}
SPL {X  -159.827, Y  +678.718, Z    +0.000, E1   +54.950, E3 -294663.517}
SPL {X  -159.222, Y  +687.156, Z    +0.000, E1   +54.792, E3 -294676.828}
SPL {X  -158.388, Y  +694.082, Z    +0.000, E1   +54.679, E3 -294687.966}
SPL {X  -157.277, Y  +700.838, Z    +0.000, E1   +54.465, E3 -294699.223}
SPL {X  -156.153, Y  +706.327, Z    +0.000, E1   +54.274, E3 -294708.559}
SPL {X  -154.917, Y  +711.470, Z    +0.000, E1   +54.052, E3 -294717.510}
SPL {X  -153.204, Y  +717.603, Z    +0.000, E1   +53.775, E3 -294728.356}
SPL {X  -151.355, Y  +723.351, Z    +0.000, E1   +53.415, E3 -294738.827}
SPL {X  -149.371, Y  +728.816, Z    +0.000, E1   +53.074, E3 -294748.918}
SPL {X  -147.376, Y  +733.767, Z    +0.000, E1   +52.671, E3 -294758.320}
SPL {X  -145.158, Y  +738.775, Z    +0.000, E1   +52.288, E3 -294767.871}
SPL {X  -142.385, Y  +744.461, Z    +0.000, E1   +51.729, E3 -294778.983}
SPL {X  -132.301, Y  +761.463, Z    +0.000, E1   +45.510, E3 -294856.722}
ENDSPLINE

SPLINE
SPL {X  -145.877, Y  +737.201, Z    +0.000, E1   +34.468, E3 -294939.833}
SPL {X  -152.550, Y  +719.721, Z    +0.000, E1   +27.728, E3 -294955.322}
SPL {X  -157.145, Y  +701.536, Z    +0.000, E1   +19.368, E3 -294964.777}
SPL {X  -159.035, Y  +688.952, Z    +0.000, E1   +12.676, E3 -294968.818}
SPL {X  -159.756, Y  +680.154, Z    +0.000, E1    +7.520, E3 -294970.544}
SPL {X  -159.986, Y  +672.560, Z    +0.000, E1    +2.636, E3 -294971.442}
SPL {X  -159.990, Y  +668.344, Z    +0.000, E1    -0.618, E3 -294971.708}
SPL {X  -159.990, Y  +664.070, Z    +0.000, E1    -5.025, E3 -294972.037}
SPL {X  -159.990, Y  +656.953, Z    +0.000, E1   -13.960, E3 -294973.103}
SPL {X  -159.990, Y  +644.589, Z    +0.000, E1   -29.011, E3 -294976.515}
SPL {X  -159.990, Y  +605.095, Z    +0.000, E1   -49.514, E3 -295001.606}
SPL {X  -159.990, Y  +546.155, Z    +0.000, E1   -54.461, E3 -295064.364}
SPL {X  -159.990, Y  +537.700, Z    +0.000, E1   -54.492, E3 -295077.128}
SPL {X  -159.990, Y  +529.394, Z    +0.000, E1   -54.464, E3 -295089.760}
SPL {X  -159.990, Y  +521.536, Z    +0.000, E1   -54.480, E3 -295101.641}
SPL {X  -159.990, Y  +514.089, Z    +0.000, E1   -54.461, E3 -295112.954}
SPL {X  -159.990, Y  +506.373, Z    +0.000, E1   -54.484, E3 -295124.590}
SPL {X  -159.990, Y  +497.571, Z    +0.000, E1   -54.478, E3 -295137.933}
SPL {X  -159.990, Y  +490.343, Z    +0.000, E1   -54.468, E3 -295148.898}
SPL {X  -159.990, Y  +483.191, Z    +0.000, E1   -54.478, E3 -295159.714}
SPL {X  -159.990, Y  +475.502, Z    +0.000, E1   -54.476, E3 -295171.364}
SPL {X  -159.990, Y  +448.520, Z    +0.000, E1   -58.543, E3 -295182.993}
SPL {X  -159.990, Y  +438.044, Z    +0.000, E1   -58.687, E3 -295195.630}
SPL {X  -159.990, Y  +431.936, Z    +0.000, E1   -57.955, E3 -295208.449}
SPL {X  -159.990, Y  +427.860, Z    +0.000, E1   -57.091, E3 -295219.513}
SPL {X  -159.990, Y  +424.653, Z    +0.000, E1   -55.901, E3 -295231.818}
SPL {X  -159.990, Y  +418.232, Z    +0.000, E1   -55.048, E3 -295246.611}
SPL {X  -159.990, Y  +410.722, Z    +0.000, E1   -54.900, E3 -295258.594}
SPL {X  -159.990, Y  +402.790, Z    +0.000, E1   -54.930, E3 -295270.369}
SPL {X  -159.990, Y  +392.953, Z    +0.000, E1   -54.918, E3 -295285.063}
SPL {X  -159.990, Y  +383.354, Z    +0.000, E1   -54.920, E3 -295299.373}
SPL {X  -159.860, Y  +376.053, Z    +0.000, E1   -54.872, E3 -295310.432}
SPL {X  -159.499, Y  +369.977, Z    +0.000, E1   -54.827, E3 -295319.837}
SPL {X  -158.803, Y  +363.045, Z    +0.000, E1   -54.709, E3 -295330.906}
SPL {X  -157.732, Y  +355.717, Z    +0.000, E1   -54.540, E3 -295342.928}
SPL {X  -156.235, Y  +348.039, Z    +0.000, E1   -54.281, E3 -295355.940}
SPL {X  -154.716, Y  +341.761, Z    +0.000, E1   -53.995, E3 -295366.897}
SPL {X  -152.882, Y  +335.340, Z    +0.000, E1   -53.695, E3 -295378.298}
SPL {X  -151.019, Y  +329.680, Z    +0.000, E1   -53.334, E3 -295388.655}
SPL {X  -149.351, Y  +325.131, Z    +0.000, E1   -53.025, E3 -295397.099}
SPL {X  -147.860, Y  +321.391, Z    +0.000, E1   -52.740, E3 -295404.152}
SPL {X  -145.914, Y  +316.881, Z    +0.000, E1   -52.402, E3 -295412.722}
SPL {X  -142.795, Y  +310.344, Z    +0.000, E1   -51.829, E3 -295425.377}
SPL {X  -132.354, Y  +292.616, Z    +0.000, E1   -44.164, E3 -295523.790}
ENDSPLINE

SPLINE
SPL {X  -150.910, Y  +329.369, Z    +0.000, E1   -29.678, E3 -295596.185}
SPL {X  -156.829, Y  +350.854, Z    +0.000, E1   -20.141, E3 -295608.738}
SPL {X  -159.049, Y  +365.169, Z    +0.000, E1   -12.580, E3 -295613.482}
SPL {X  -159.776, Y  +374.231, Z    +0.000, E1    -7.281, E3 -295615.368}
SPL {X  -159.986, Y  +381.380, Z    +0.000, E1    -2.685, E3 -295616.214}
SPL {X  -159.990, Y  +384.493, Z    +0.000, E1    -0.324, E3 -295616.422}
SPL {X  -159.990, Y  +387.327, Z    +0.000, E1    +2.137, E3 -295616.605}
SPL {X  -159.990, Y  +392.053, Z    +0.000, E1    +7.477, E3 -295617.070}
SPL {X  -159.990, Y  +396.158, Z    +0.000, E1   +12.775, E3 -295617.695}
SPL {X  -159.990, Y  +401.377, Z    +0.000, E1   +19.398, E3 -295618.876}
SPL {X  -159.990, Y  +411.365, Z    +0.000, E1   +30.630, E3 -295622.084}
SPL {X  -159.990, Y  +450.467, Z    +0.000, E1   +50.183, E3 -295645.733}
SPL {X  -159.990, Y  +509.934, Z    +0.000, E1   +54.923, E3 -295708.352}
SPL {X  -159.990, Y  +516.848, Z    +0.000, E1   +54.930, E3 -295718.640}
SPL {X  -159.990, Y  +524.818, Z    +0.000, E1   +54.933, E3 -295730.512}
SPL {X  -159.990, Y  +532.100, Z    +0.000, E1   +54.924, E3 -295741.365}
SPL {X  -159.990, Y  +539.391, Z    +0.000, E1   +54.933, E3 -295752.217}
SPL {X  -159.990, Y  +546.283, Z    +0.000, E1   +54.924, E3 -295762.488}
SPL {X  -159.990, Y  +553.734, Z    +0.000, E1   +54.938, E3 -295773.575}
SPL {X  -159.990, Y  +560.983, Z    +0.000, E1   +54.918, E3 -295784.413}
SPL {X  -159.990, Y  +567.462, Z    +0.000, E1   +54.929, E3 -295794.048}
SPL {X  -159.990, Y  +575.140, Z    +0.000, E1   +54.928, E3 -295805.480}
SPL {X  -159.990, Y  +581.046, Z    +0.000, E1   +54.920, E3 -295814.292}
SPL {X  -159.990, Y  +588.063, Z    +0.000, E1   +54.931, E3 -295824.727}
SPL {X  -159.990, Y  +595.273, Z    +0.000, E1   +54.928, E3 -295835.451}
SPL {X  -159.990, Y  +602.326, Z    +0.000, E1   +54.932, E3 -295845.951}
SPL {X  -159.990, Y  +610.296, Z    +0.000, E1   +54.937, E3 -295857.820}
SPL {X  -159.990, Y  +618.534, Z    +0.000, E1   +54.942, E3 -295870.057}
SPL {X  -159.990, Y  +625.928, Z    +0.000, E1   +54.931, E3 -295881.083}
SPL {X  -159.990, Y  +633.423, Z    +0.000, E1   +54.943, E3 -295892.225}
SPL {X  -159.990, Y  +643.352, Z    +0.000, E1   +54.966, E3 -295906.960}
SPL {X  -159.990, Y  +650.756, Z    +0.000, E1   +54.931, E3 -295918.027}
SPL {X  -159.990, Y  +658.525, Z    +0.000, E1   +54.959, E3 -295929.563}
SPL {X  -159.990, Y  +667.903, Z    +0.000, E1   +54.941, E3 -295943.594}
SPL {X  -159.953, Y  +674.920, Z    +0.000, E1   +54.918, E3 -295954.097}
SPL {X  -159.714, Y  +680.893, Z    +0.000, E1   +54.890, E3 -295963.237}
SPL {X  -159.222, Y  +687.156, Z    +0.000, E1   +54.792, E3 -295973.124}
SPL {X  -158.388, Y  +694.082, Z    +0.000, E1   +54.679, E3 -295984.262}
SPL {X  -157.277, Y  +700.838, Z    +0.000, E1   +54.465, E3 -295995.519}
SPL {X  -156.153, Y  +706.327, Z    +0.000, E1   +54.274, E3 -296004.855}
SPL {X  -154.917, Y  +711.470, Z    +0.000, E1   +54.052, E3 -296013.806}
SPL {X  -153.204, Y  +717.603, Z    +0.000, E1   +53.775, E3 -296024.652}
SPL {X  -151.355, Y  +723.351, Z    +0.000, E1   +53.415, E3 -296035.124}
SPL {X  -149.371, Y  +728.816, Z    +0.000, E1   +53.074, E3 -296045.214}
SPL {X  -146.631, Y  +735.501, Z    +0.000, E1   +52.568, E3 -296057.875}
SPL {X  -144.428, Y  +740.329, Z    +0.000, E1   +52.109, E3 -296067.229}
SPL {X  -142.385, Y  +744.461, Z    +0.000, E1   +51.729, E3 -296075.280}
SPL {X  -132.301, Y  +761.463, Z    +0.000, E1   +45.510, E3 -296153.018}
ENDSPLINE

SPLINE
SPL {X  -145.877, Y  +737.201, Z    +0.000, E1   +34.468, E3 -296236.129}
SPL {X  -152.550, Y  +719.721, Z    +0.000, E1   +27.728, E3 -296251.618}
SPL {X  -157.145, Y  +701.536, Z    +0.000, E1   +19.368, E3 -296261.073}
SPL {X  -159.035, Y  +688.952, Z    +0.000, E1   +12.676, E3 -296265.114}
SPL {X  -159.756, Y  +680.154, Z    +0.000, E1    +7.520, E3 -296266.840}
SPL {X  -159.986, Y  +672.560, Z    +0.000, E1    +2.636, E3 -296267.738}
SPL {X  -159.990, Y  +668.344, Z    +0.000, E1    -0.618, E3 -296268.005}
SPL {X  -159.990, Y  +664.070, Z    +0.000, E1    -5.025, E3 -296268.333}
SPL {X  -159.990, Y  +656.953, Z    +0.000, E1   -13.960, E3 -296269.400}
SPL {X  -159.990, Y  +644.589, Z    +0.000, E1   -29.011, E3 -296272.811}
SPL {X  -159.990, Y  +605.095, Z    +0.000, E1   -49.514, E3 -296297.902}
SPL {X  -159.990, Y  +543.998, Z    +0.000, E1   -54.483, E3 -296363.892}
SPL {X  -159.990, Y  +535.878, Z    +0.000, E1   -54.465, E3 -296376.226}
SPL {X  -159.990, Y  +529.394, Z    +0.000, E1   -54.464, E3 -296386.056}
SPL {X  -159.990, Y  +521.536, Z    +0.000, E1   -54.480, E3 -296397.938}
SPL {X  -159.990, Y  +514.089, Z    +0.000, E1   -54.461, E3 -296409.250}
SPL {X  -159.990, Y  +506.373, Z    +0.000, E1   -54.484, E3 -296420.886}
SPL {X  -159.990, Y  +497.571, Z    +0.000, E1   -54.478, E3 -296434.230}
SPL {X  -159.990, Y  +490.343, Z    +0.000, E1   -54.468, E3 -296445.195}
SPL {X  -159.990, Y  +483.191, Z    +0.000, E1   -54.478, E3 -296456.011}
SPL {X  -159.990, Y  +475.502, Z    +0.000, E1   -54.476, E3 -296467.660}
SPL {X  -159.990, Y  +448.520, Z    +0.000, E1   -58.543, E3 -296479.289}
SPL {X  -159.990, Y  +438.044, Z    +0.000, E1   -58.687, E3 -296491.926}
SPL {X  -159.990, Y  +431.936, Z    +0.000, E1   -57.955, E3 -296504.745}
SPL {X  -159.990, Y  +427.860, Z    +0.000, E1   -57.091, E3 -296515.809}
SPL {X  -159.990, Y  +424.653, Z    +0.000, E1   -55.901, E3 -296528.114}
SPL {X  -159.990, Y  +418.232, Z    +0.000, E1   -55.048, E3 -296542.907}
SPL {X  -159.990, Y  +410.722, Z    +0.000, E1   -54.900, E3 -296554.890}
SPL {X  -159.990, Y  +402.790, Z    +0.000, E1   -54.930, E3 -296566.665}
SPL {X  -159.990, Y  +392.953, Z    +0.000, E1   -54.918, E3 -296581.359}
SPL {X  -159.990, Y  +383.354, Z    +0.000, E1   -54.920, E3 -296595.669}
SPL {X  -159.860, Y  +376.053, Z    +0.000, E1   -54.872, E3 -296606.729}
SPL {X  -159.499, Y  +369.977, Z    +0.000, E1   -54.827, E3 -296616.133}
SPL {X  -158.803, Y  +363.045, Z    +0.000, E1   -54.709, E3 -296627.202}
SPL {X  -157.966, Y  +357.131, Z    +0.000, E1   -54.559, E3 -296636.905}
SPL {X  -156.775, Y  +350.586, Z    +0.000, E1   -54.373, E3 -296647.879}
SPL {X  -155.027, Y  +342.959, Z    +0.000, E1   -54.074, E3 -296661.052}
SPL {X  -153.580, Y  +337.668, Z    +0.000, E1   -53.781, E3 -296670.475}
SPL {X  -151.643, Y  +331.497, Z    +0.000, E1   -53.493, E3 -296681.554}
SPL {X  -149.351, Y  +325.131, Z    +0.000, E1   -53.025, E3 -296693.396}
SPL {X  -147.860, Y  +321.391, Z    +0.000, E1   -52.740, E3 -296700.448}
SPL {X  -145.914, Y  +316.881, Z    +0.000, E1   -52.402, E3 -296709.018}
SPL {X  -142.795, Y  +310.344, Z    +0.000, E1   -51.829, E3 -296721.674}
SPL {X  -132.354, Y  +292.616, Z    +0.000, E1   -44.164, E3 -296820.086}
ENDSPLINE

SPLINE
SPL {X  -150.910, Y  +329.369, Z    +0.000, E1   -29.678, E3 -296892.481}
SPL {X  -156.829, Y  +350.854, Z    +0.000, E1   -20.141, E3 -296905.034}
SPL {X  -159.049, Y  +365.169, Z    +0.000, E1   -12.580, E3 -296909.778}
SPL {X  -159.881, Y  +376.607, Z    +0.000, E1    -5.865, E3 -296911.988}
SPL {X  -159.990, Y  +382.403, Z    +0.000, E1    -1.910, E3 -296912.593}
SPL {X  -159.990, Y  +385.261, Z    +0.000, E1    +0.259, E3 -296912.764}
SPL {X  -159.990, Y  +388.094, Z    +0.000, E1    +3.012, E3 -296912.956}
SPL {X  -159.990, Y  +392.053, Z    +0.000, E1    +7.477, E3 -296913.366}
SPL {X  -159.990, Y  +396.158, Z    +0.000, E1   +12.775, E3 -296913.992}
SPL {X  -159.990, Y  +401.377, Z    +0.000, E1   +19.398, E3 -296915.172}
SPL {X  -159.990, Y  +411.365, Z    +0.000, E1   +30.630, E3 -296918.380}
SPL {X  -159.990, Y  +450.467, Z    +0.000, E1   +50.183, E3 -296942.029}
SPL {X  -159.990, Y  +509.934, Z    +0.000, E1   +54.923, E3 -297004.648}
SPL {X  -159.990, Y  +516.848, Z    +0.000, E1   +54.930, E3 -297014.936}
SPL {X  -159.990, Y  +524.818, Z    +0.000, E1   +54.933, E3 -297026.808}
SPL {X  -159.990, Y  +532.100, Z    +0.000, E1   +54.924, E3 -297037.661}
SPL {X  -159.990, Y  +539.391, Z    +0.000, E1   +54.933, E3 -297048.513}
SPL {X  -159.990, Y  +546.283, Z    +0.000, E1   +54.924, E3 -297058.785}
SPL {X  -159.990, Y  +553.734, Z    +0.000, E1   +54.938, E3 -297069.871}
SPL {X  -159.990, Y  +564.956, Z    +0.000, E1   +54.973, E3 -297086.543}
SPL {X  -159.990, Y  +577.902, Z    +0.000, E1   +54.969, E3 -297105.833}
SPL {X  -159.990, Y  +588.063, Z    +0.000, E1   +54.931, E3 -297121.023}
SPL {X  -159.990, Y  +595.273, Z    +0.000, E1   +54.928, E3 -297131.747}
SPL {X  -159.990, Y  +602.326, Z    +0.000, E1   +54.932, E3 -297142.247}
SPL {X  -159.990, Y  +610.296, Z    +0.000, E1   +54.937, E3 -297154.117}
SPL {X  -159.990, Y  +618.534, Z    +0.000, E1   +54.942, E3 -297166.354}
SPL {X  -159.990, Y  +625.928, Z    +0.000, E1   +54.931, E3 -297177.379}
SPL {X  -159.990, Y  +633.423, Z    +0.000, E1   +54.943, E3 -297188.521}
SPL {X  -159.990, Y  +640.333, Z    +0.000, E1   +54.927, E3 -297198.835}
SPL {X  -159.990, Y  +648.272, Z    +0.000, E1   +54.961, E3 -297210.583}
SPL {X  -159.990, Y  +655.990, Z    +0.000, E1   +54.930, E3 -297222.130}
SPL {X  -159.990, Y  +665.734, Z    +0.000, E1   +54.984, E3 -297236.581}
SPL {X  -159.827, Y  +678.718, Z    +0.000, E1   +54.950, E3 -297256.110}
SPL {X  -159.222, Y  +687.156, Z    +0.000, E1   +54.792, E3 -297269.420}
SPL {X  -158.388, Y  +694.082, Z    +0.000, E1   +54.679, E3 -297280.558}
SPL {X  -157.277, Y  +700.838, Z    +0.000, E1   +54.465, E3 -297291.815}
SPL {X  -156.153, Y  +706.327, Z    +0.000, E1   +54.274, E3 -297301.151}
SPL {X  -154.917, Y  +711.470, Z    +0.000, E1   +54.052, E3 -297310.103}
SPL {X  -153.204, Y  +717.603, Z    +0.000, E1   +53.775, E3 -297320.949}
SPL {X  -151.355, Y  +723.351, Z    +0.000, E1   +53.415, E3 -297331.420}
SPL {X  -149.371, Y  +728.816, Z    +0.000, E1   +53.074, E3 -297341.511}
SPL {X  -147.376, Y  +733.767, Z    +0.000, E1   +52.671, E3 -297350.913}
SPL {X  -145.158, Y  +738.775, Z    +0.000, E1   +52.288, E3 -297360.464}
SPL {X  -142.385, Y  +744.461, Z    +0.000, E1   +51.729, E3 -297371.576}
SPL {X  -132.301, Y  +761.463, Z    +0.000, E1   +45.510, E3 -297449.315}
ENDSPLINE

SPLINE
SPL {X  -145.877, Y  +737.201, Z    +0.000, E1   +34.468, E3 -297532.425}
SPL {X  -152.550, Y  +719.721, Z    +0.000, E1   +27.728, E3 -297547.915}
SPL {X  -157.145, Y  +701.536, Z    +0.000, E1   +19.368, E3 -297557.369}
SPL {X  -159.035, Y  +688.952, Z    +0.000, E1   +12.676, E3 -297561.410}
SPL {X  -159.756, Y  +680.154, Z    +0.000, E1    +7.520, E3 -297563.137}
SPL {X  -159.986, Y  +672.560, Z    +0.000, E1    +2.636, E3 -297564.035}
SPL {X  -159.990, Y  +668.344, Z    +0.000, E1    -0.618, E3 -297564.301}
SPL {X  -159.990, Y  +664.070, Z    +0.000, E1    -5.025, E3 -297564.629}
SPL {X  -159.990, Y  +658.737, Z    +0.000, E1   -11.801, E3 -297565.336}
SPL {X  -159.990, Y  +652.023, Z    +0.000, E1   -20.449, E3 -297566.820}
SPL {X  -159.990, Y  +641.935, Z    +0.000, E1   -31.848, E3 -297569.992}
SPL {X  -159.990, Y  +605.095, Z    +0.000, E1   -49.514, E3 -297594.198}
SPL {X  -159.990, Y  +543.998, Z    +0.000, E1   -54.483, E3 -297660.188}
SPL {X  -159.990, Y  +535.878, Z    +0.000, E1   -54.465, E3 -297672.523}
SPL {X  -159.990, Y  +529.394, Z    +0.000, E1   -54.464, E3 -297682.352}
SPL {X  -159.990, Y  +521.536, Z    +0.000, E1   -54.480, E3 -297694.234}
SPL {X  -159.990, Y  +514.089, Z    +0.000, E1   -54.461, E3 -297705.546}
SPL {X  -159.990, Y  +506.373, Z    +0.000, E1   -54.484, E3 -297717.183}
SPL {X  -159.990, Y  +497.571, Z    +0.000, E1   -54.478, E3 -297730.526}
SPL {X  -159.990, Y  +490.343, Z    +0.000, E1   -54.468, E3 -297741.491}
SPL {X  -159.990, Y  +483.191, Z    +0.000, E1   -54.478, E3 -297752.307}
SPL {X  -159.990, Y  +475.502, Z    +0.000, E1   -54.476, E3 -297763.956}
SPL {X  -159.990, Y  +448.520, Z    +0.000, E1   -58.543, E3 -297775.585}
SPL {X  -159.990, Y  +438.044, Z    +0.000, E1   -58.687, E3 -297788.222}
SPL {X  -159.990, Y  +431.936, Z    +0.000, E1   -57.955, E3 -297801.042}
SPL {X  -159.990, Y  +427.860, Z    +0.000, E1   -57.091, E3 -297812.105}
SPL {X  -159.990, Y  +424.653, Z    +0.000, E1   -55.901, E3 -297824.411}
SPL {X  -159.990, Y  +418.232, Z    +0.000, E1   -55.048, E3 -297839.204}
SPL {X  -159.990, Y  +410.722, Z    +0.000, E1   -54.900, E3 -297851.187}
SPL {X  -159.990, Y  +402.790, Z    +0.000, E1   -54.930, E3 -297862.962}
SPL {X  -159.990, Y  +391.119, Z    +0.000, E1   -54.948, E3 -297880.339}
SPL {X  -159.988, Y  +381.720, Z    +0.000, E1   -54.897, E3 -297894.447}
SPL {X  -159.769, Y  +374.091, Z    +0.000, E1   -54.882, E3 -297905.998}
SPL {X  -158.996, Y  +364.689, Z    +0.000, E1   -54.773, E3 -297920.794}
SPL {X  -157.966, Y  +357.131, Z    +0.000, E1   -54.559, E3 -297933.201}
SPL {X  -156.481, Y  +349.175, Z    +0.000, E1   -54.353, E3 -297946.541}
SPL {X  -154.716, Y  +341.761, Z    +0.000, E1   -53.995, E3 -297959.489}
SPL {X  -152.882, Y  +335.340, Z    +0.000, E1   -53.695, E3 -297970.891}
SPL {X  -151.019, Y  +329.680, Z    +0.000, E1   -53.334, E3 -297981.248}
SPL {X  -149.351, Y  +325.131, Z    +0.000, E1   -53.025, E3 -297989.692}
SPL {X  -147.860, Y  +321.391, Z    +0.000, E1   -52.740, E3 -297996.744}
SPL {X  -145.914, Y  +316.881, Z    +0.000, E1   -52.402, E3 -298005.314}
SPL {X  -142.795, Y  +310.344, Z    +0.000, E1   -51.829, E3 -298017.970}
SPL {X  -132.354, Y  +292.616, Z    +0.000, E1   -44.164, E3 -298116.382}
ENDSPLINE

SPLINE
SPL {X  -150.910, Y  +329.369, Z    +0.000, E1   -29.678, E3 -298188.778}
SPL {X  -156.396, Y  +348.778, Z    +0.000, E1   -21.134, E3 -298200.421}
SPL {X  -158.554, Y  +361.116, Z    +0.000, E1   -14.883, E3 -298204.875}
SPL {X  -159.881, Y  +376.607, Z    +0.000, E1    -5.865, E3 -298208.284}
SPL {X  -159.990, Y  +383.659, Z    +0.000, E1    -1.050, E3 -298208.965}
SPL {X  -159.990, Y  +387.327, Z    +0.000, E1    +2.137, E3 -298209.197}
SPL {X  -159.990, Y  +390.622, Z    +0.000, E1    +5.876, E3 -298209.491}
SPL {X  -159.990, Y  +394.493, Z    +0.000, E1   +10.512, E3 -298210.014}
SPL {X  -159.990, Y  +401.377, Z    +0.000, E1   +19.398, E3 -298211.468}
SPL {X  -159.990, Y  +411.365, Z    +0.000, E1   +30.630, E3 -298214.677}
SPL {X  -159.990, Y  +450.467, Z    +0.000, E1   +50.183, E3 -298238.326}
SPL {X  -159.990, Y  +509.934, Z    +0.000, E1   +54.923, E3 -298300.944}
SPL {X  -159.990, Y  +516.848, Z    +0.000, E1   +54.930, E3 -298311.232}
SPL {X  -159.990, Y  +524.818, Z    +0.000, E1   +54.933, E3 -298323.104}
SPL {X  -159.990, Y  +532.100, Z    +0.000, E1   +54.924, E3 -298333.957}
SPL {X  -159.990, Y  +539.391, Z    +0.000, E1   +54.933, E3 -298344.809}
SPL {X  -159.990, Y  +546.283, Z    +0.000, E1   +54.924, E3 -298355.081}
SPL {X  -159.990, Y  +553.734, Z    +0.000, E1   +54.938, E3 -298366.168}
SPL {X  -159.990, Y  +560.983, Z    +0.000, E1   +54.918, E3 -298377.005}
SPL {X  -159.990, Y  +567.462, Z    +0.000, E1   +54.929, E3 -298386.640}
SPL {X  -159.990, Y  +575.140, Z    +0.000, E1   +54.928, E3 -298398.072}
SPL {X  -159.990, Y  +581.046, Z    +0.000, E1   +54.920, E3 -298406.885}
SPL {X  -159.990, Y  +588.063, Z    +0.000, E1   +54.931, E3 -298417.320}
SPL {X  -159.990, Y  +595.273, Z    +0.000, E1   +54.928, E3 -298428.043}
SPL {X  -159.990, Y  +602.326, Z    +0.000, E1   +54.932, E3 -298438.544}
SPL {X  -159.990, Y  +610.296, Z    +0.000, E1   +54.937, E3 -298450.413}
SPL {X  -159.990, Y  +618.534, Z    +0.000, E1   +54.942, E3 -298462.650}
SPL {X  -159.990, Y  +628.178, Z    +0.000, E1   +54.959, E3 -298476.981}
SPL {X  -159.990, Y  +638.304, Z    +0.000, E1   +54.952, E3 -298492.070}
SPL {X  -159.990, Y  +645.976, Z    +0.000, E1   +54.934, E3 -298503.504}
SPL {X  -159.990, Y  +653.679, Z    +0.000, E1   +54.961, E3 -298514.929}
SPL {X  -159.990, Y  +665.734, Z    +0.000, E1   +54.984, E3 -298532.878}
SPL {X  -159.827, Y  +678.718, Z    +0.000, E1   +54.950, E3 -298552.406}
SPL {X  -159.222, Y  +687.156, Z    +0.000, E1   +54.792, E3 -298565.717}
SPL {X  -158.388, Y  +694.082, Z    +0.000, E1   +54.679, E3 -298576.854}
SPL {X  -157.277, Y  +700.838, Z    +0.000, E1   +54.465, E3 -298588.112}
SPL {X  -156.153, Y  +706.327, Z    +0.000, E1   +54.274, E3 -298597.448}
SPL {X  -154.917, Y  +711.470, Z    +0.000, E1   +54.052, E3 -298606.399}
SPL {X  -153.204, Y  +717.603, Z    +0.000, E1   +53.775, E3 -298617.245}
SPL {X  -151.355, Y  +723.351, Z    +0.000, E1   +53.415, E3 -298627.716}
SPL {X  -149.371, Y  +728.816, Z    +0.000, E1   +53.074, E3 -298637.807}
SPL {X  -146.631, Y  +735.501, Z    +0.000, E1   +52.568, E3 -298650.467}
SPL {X  -144.428, Y  +740.329, Z    +0.000, E1   +52.109, E3 -298659.821}
SPL {X  -142.385, Y  +744.461, Z    +0.000, E1   +51.729, E3 -298667.872}
SPL {X  -132.301, Y  +761.463, Z    +0.000, E1   +45.510, E3 -298745.611}
ENDSPLINE

SPLINE
SPL {X  -145.877, Y  +737.201, Z    +0.000, E1   +34.468, E3 -298828.722}
SPL {X  -152.550, Y  +719.721, Z    +0.000, E1   +27.728, E3 -298844.211}
SPL {X  -157.145, Y  +701.536, Z    +0.000, E1   +19.368, E3 -298853.666}
SPL {X  -159.035, Y  +688.952, Z    +0.000, E1   +12.676, E3 -298857.707}
SPL {X  -159.756, Y  +680.154, Z    +0.000, E1    +7.520, E3 -298859.433}
SPL {X  -159.986, Y  +672.560, Z    +0.000, E1    +2.636, E3 -298860.331}
SPL {X  -159.990, Y  +668.344, Z    +0.000, E1    -0.618, E3 -298860.597}
SPL {X  -159.990, Y  +664.070, Z    +0.000, E1    -5.025, E3 -298860.926}
SPL {X  -159.990, Y  +656.953, Z    +0.000, E1   -13.960, E3 -298861.992}
SPL {X  -159.990, Y  +644.589, Z    +0.000, E1   -29.011, E3 -298865.404}
SPL {X  -159.990, Y  +605.095, Z    +0.000, E1   -49.514, E3 -298890.495}
SPL {X  -159.990, Y  +543.998, Z    +0.000, E1   -54.483, E3 -298956.484}
SPL {X  -159.990, Y  +535.878, Z    +0.000, E1   -54.465, E3 -298968.819}
SPL {X  -159.990, Y  +529.394, Z    +0.000, E1   -54.464, E3 -298978.649}
SPL {X  -159.990, Y  +521.536, Z    +0.000, E1   -54.480, E3 -298990.530}
SPL {X  -159.990, Y  +514.089, Z    +0.000, E1   -54.461, E3 -299001.843}
SPL {X  -159.990, Y  +506.373, Z    +0.000, E1   -54.484, E3 -299013.479}
SPL {X  -159.990, Y  +497.571, Z    +0.000, E1   -54.478, E3 -299026.822}
SPL {X  -159.990, Y  +490.343, Z    +0.000, E1   -54.468, E3 -299037.787}
SPL {X  -159.990, Y  +483.191, Z    +0.000, E1   -54.478, E3 -299048.603}
SPL {X  -159.990, Y  +475.502, Z    +0.000, E1   -54.476, E3 -299060.253}
SPL {X  -159.990, Y  +448.520, Z    +0.000, E1   -58.543, E3 -299071.882}
SPL {X  -159.990, Y  +438.044, Z    +0.000, E1   -58.687, E3 -299084.518}
SPL {X  -159.990, Y  +431.936, Z    +0.000, E1   -57.955, E3 -299097.338}
SPL {X  -159.990, Y  +427.293, Z    +0.000, E1   -56.830, E3 -299111.044}
SPL {X  -159.990, Y  +423.841, Z    +0.000, E1   -55.679, E3 -299123.146}
SPL {X  -159.990, Y  +418.232, Z    +0.000, E1   -55.048, E3 -299135.500}
SPL {X  -159.990, Y  +410.722, Z    +0.000, E1   -54.900, E3 -299147.483}
SPL {X  -159.990, Y  +402.790, Z    +0.000, E1   -54.930, E3 -299159.258}
SPL {X  -159.990, Y  +392.953, Z    +0.000, E1   -54.918, E3 -299173.952}
SPL {X  -159.990, Y  +383.354, Z    +0.000, E1   -54.920, E3 -299188.262}
SPL {X  -159.660, Y  +372.225, Z    +0.000, E1   -54.896, E3 -299205.143}
SPL {X  -158.803, Y  +363.045, Z    +0.000, E1   -54.709, E3 -299219.795}
SPL {X  -157.732, Y  +355.717, Z    +0.000, E1   -54.540, E3 -299231.817}
SPL {X  -156.235, Y  +348.039, Z    +0.000, E1   -54.281, E3 -299244.829}
SPL {X  -154.716, Y  +341.761, Z    +0.000, E1   -53.995, E3 -299255.785}
SPL {X  -152.882, Y  +335.340, Z    +0.000, E1   -53.695, E3 -299267.187}
SPL {X  -151.019, Y  +329.680, Z    +0.000, E1   -53.334, E3 -299277.544}
SPL {X  -148.682, Y  +323.421, Z    +0.000, E1   -52.939, E3 -299289.146}
SPL {X  -145.914, Y  +316.881, Z    +0.000, E1   -52.402, E3 -299301.611}
SPL {X  -142.795, Y  +310.344, Z    +0.000, E1   -51.829, E3 -299314.266}
SPL {X  -132.354, Y  +292.616, Z    +0.000, E1   -44.164, E3 -299412.679}
ENDSPLINE

SPLINE
SPL {X  -150.910, Y  +329.369, Z    +0.000, E1   -29.678, E3 -299485.074}
SPL {X  -156.829, Y  +350.854, Z    +0.000, E1   -20.141, E3 -299497.627}
SPL {X  -159.049, Y  +365.169, Z    +0.000, E1   -12.580, E3 -299502.371}
SPL {X  -159.776, Y  +374.231, Z    +0.000, E1    -7.281, E3 -299504.257}
SPL {X  -159.986, Y  +381.380, Z    +0.000, E1    -2.685, E3 -299505.103}
SPL {X  -159.990, Y  +384.493, Z    +0.000, E1    -0.324, E3 -299505.311}
SPL {X  -159.990, Y  +387.327, Z    +0.000, E1    +2.137, E3 -299505.494}
SPL {X  -159.990, Y  +390.622, Z    +0.000, E1    +5.876, E3 -299505.787}
SPL {X  -159.990, Y  +394.493, Z    +0.000, E1   +10.512, E3 -299506.310}
SPL {X  -159.990, Y  +401.377, Z    +0.000, E1   +19.398, E3 -299507.765}
SPL {X  -159.990, Y  +411.365, Z    +0.000, E1   +30.630, E3 -299510.973}
SPL {X  -159.990, Y  +450.467, Z    +0.000, E1   +50.183, E3 -299534.622}
SPL {X  -159.990, Y  +509.934, Z    +0.000, E1   +54.923, E3 -299597.241}
SPL {X  -159.990, Y  +516.848, Z    +0.000, E1   +54.930, E3 -299607.529}
SPL {X  -159.990, Y  +524.818, Z    +0.000, E1   +54.933, E3 -299619.401}
SPL {X  -159.990, Y  +532.100, Z    +0.000, E1   +54.924, E3 -299630.254}
SPL {X  -159.990, Y  +539.391, Z    +0.000, E1   +54.933, E3 -299641.106}
SPL {X  -159.990, Y  +546.283, Z    +0.000, E1   +54.924, E3 -299651.377}
SPL {X  -159.990, Y  +553.734, Z    +0.000, E1   +54.938, E3 -299662.464}
SPL {X  -159.990, Y  +560.983, Z    +0.000, E1   +54.918, E3 -299673.301}
SPL {X  -159.990, Y  +567.462, Z    +0.000, E1   +54.929, E3 -299682.936}
SPL {X  -159.990, Y  +575.140, Z    +0.000, E1   +54.928, E3 -299694.369}
SPL {X  -159.990, Y  +581.046, Z    +0.000, E1   +54.920, E3 -299703.181}
SPL {X  -159.990, Y  +588.063, Z    +0.000, E1   +54.931, E3 -299713.616}
SPL {X  -159.990, Y  +595.273, Z    +0.000, E1   +54.928, E3 -299724.339}
SPL {X  -159.990, Y  +602.326, Z    +0.000, E1   +54.932, E3 -299734.840}
SPL {X  -159.990, Y  +610.296, Z    +0.000, E1   +54.937, E3 -299746.709}
SPL {X  -159.990, Y  +618.534, Z    +0.000, E1   +54.942, E3 -299758.946}
SPL {X  -159.990, Y  +628.178, Z    +0.000, E1   +54.959, E3 -299773.277}
SPL {X  -159.990, Y  +638.304, Z    +0.000, E1   +54.952, E3 -299788.366}
SPL {X  -159.990, Y  +648.272, Z    +0.000, E1   +54.961, E3 -299803.175}
SPL {X  -159.990, Y  +655.990, Z    +0.000, E1   +54.930, E3 -299814.723}
SPL {X  -159.990, Y  +665.734, Z    +0.000, E1   +54.984, E3 -299829.174}
SPL {X  -159.953, Y  +674.920, Z    +0.000, E1   +54.918, E3 -299842.986}
SPL {X  -159.714, Y  +680.893, Z    +0.000, E1   +54.890, E3 -299852.126}
SPL {X  -158.975, Y  +689.491, Z    +0.000, E1   +54.786, E3 -299865.691}
SPL {X  -157.608, Y  +699.005, Z    +0.000, E1   +54.556, E3 -299881.285}
SPL {X  -156.153, Y  +706.327, Z    +0.000, E1   +54.274, E3 -299893.744}
SPL {X  -154.917, Y  +711.470, Z    +0.000, E1   +54.052, E3 -299902.695}
SPL {X  -153.204, Y  +717.603, Z    +0.000, E1   +53.775, E3 -299913.541}
SPL {X  -150.773, Y  +725.019, Z    +0.000, E1   +53.343, E3 -299927.034}
SPL {X  -148.029, Y  +732.198, Z    +0.000, E1   +52.831, E3 -299940.471}
SPL {X  -145.158, Y  +738.775, Z    +0.000, E1   +52.288, E3 -299953.057}
SPL {X  -142.385, Y  +744.461, Z    +0.000, E1   +51.729, E3 -299964.169}
SPL {X  -132.301, Y  +761.463, Z    +0.000, E1   +45.510, E3 -300041.907}
ENDSPLINE

SPLINE
SPL {X  -145.877, Y  +737.201, Z    +0.000, E1   +34.468, E3 -300125.018}
SPL {X  -152.550, Y  +719.721, Z    +0.000, E1   +27.728, E3 -300140.507}
SPL {X  -157.145, Y  +701.536, Z    +0.000, E1   +19.368, E3 -300149.962}
SPL {X  -159.035, Y  +688.952, Z    +0.000, E1   +12.676, E3 -300154.003}
SPL {X  -159.873, Y  +677.622, Z    +0.000, E1    +6.008, E3 -300156.075}
SPL {X  -159.990, Y  +670.381, Z    +0.000, E1    +1.064, E3 -300156.775}
SPL {X  -159.990, Y  +666.603, Z    +0.000, E1    -2.256, E3 -300157.007}
SPL {X  -159.990, Y  +662.759, Z    +0.000, E1    -6.725, E3 -300157.350}
SPL {X  -159.990, Y  +658.737, Z    +0.000, E1   -11.801, E3 -300157.928}
SPL {X  -159.990, Y  +652.023, Z    +0.000, E1   -20.449, E3 -300159.412}
SPL {X  -159.990, Y  +641.935, Z    +0.000, E1   -31.848, E3 -300162.584}
SPL {X  -159.990, Y  +605.095, Z    +0.000, E1   -49.514, E3 -300186.791}
SPL {X  -159.990, Y  +543.998, Z    +0.000, E1   -54.483, E3 -300252.781}
SPL {X  -159.990, Y  +535.878, Z    +0.000, E1   -54.465, E3 -300265.115}
SPL {X  -159.990, Y  +529.394, Z    +0.000, E1   -54.464, E3 -300274.945}
SPL {X  -159.990, Y  +521.536, Z    +0.000, E1   -54.480, E3 -300286.827}
SPL {X  -159.990, Y  +514.089, Z    +0.000, E1   -54.461, E3 -300298.139}
SPL {X  -159.990, Y  +506.373, Z    +0.000, E1   -54.484, E3 -300309.775}
SPL {X  -159.990, Y  +497.571, Z    +0.000, E1   -54.478, E3 -300323.118}
SPL {X  -159.990, Y  +490.343, Z    +0.000, E1   -54.468, E3 -300334.084}
SPL {X  -159.990, Y  +483.191, Z    +0.000, E1   -54.478, E3 -300344.900}
SPL {X  -159.990, Y  +475.502, Z    +0.000, E1   -54.476, E3 -300356.549}
SPL {X  -159.990, Y  +448.520, Z    +0.000, E1   -58.543, E3 -300368.178}
SPL {X  -159.990, Y  +438.044, Z    +0.000, E1   -58.687, E3 -300380.815}
SPL {X  -159.990, Y  +431.936, Z    +0.000, E1   -57.955, E3 -300393.634}
SPL {X  -159.990, Y  +427.293, Z    +0.000, E1   -56.830, E3 -300407.340}
SPL {X  -159.990, Y  +423.841, Z    +0.000, E1   -55.679, E3 -300419.442}
SPL {X  -159.990, Y  +418.232, Z    +0.000, E1   -55.048, E3 -300431.796}
SPL {X  -159.990, Y  +407.911, Z    +0.000, E1   -54.938, E3 -300447.910}
SPL {X  -159.990, Y  +400.284, Z    +0.000, E1   -54.897, E3 -300459.343}
SPL {X  -159.990, Y  +392.953, Z    +0.000, E1   -54.918, E3 -300470.248}
SPL {X  -159.990, Y  +383.354, Z    +0.000, E1   -54.920, E3 -300484.558}
SPL {X  -159.660, Y  +372.225, Z    +0.000, E1   -54.896, E3 -300501.439}
SPL {X  -158.803, Y  +363.045, Z    +0.000, E1   -54.709, E3 -300516.091}
SPL {X  -157.966, Y  +357.131, Z    +0.000, E1   -54.559, E3 -300525.794}
SPL {X  -156.481, Y  +349.175, Z    +0.000, E1   -54.353, E3 -300539.133}
SPL {X  -154.716, Y  +341.761, Z    +0.000, E1   -53.995, E3 -300552.082}
SPL {X  -152.882, Y  +335.340, Z    +0.000, E1   -53.695, E3 -300563.483}
SPL {X  -151.019, Y  +329.680, Z    +0.000, E1   -53.334, E3 -300573.840}
SPL {X  -148.682, Y  +323.421, Z    +0.000, E1   -52.939, E3 -300585.443}
SPL {X  -145.914, Y  +316.881, Z    +0.000, E1   -52.402, E3 -300597.907}
SPL {X  -142.795, Y  +310.344, Z    +0.000, E1   -51.829, E3 -300610.563}
SPL {X  -132.354, Y  +292.616, Z    +0.000, E1   -44.164, E3 -300708.975}
ENDSPLINE

SPLINE
SPL {X  -150.910, Y  +329.369, Z    +0.000, E1   -29.678, E3 -300781.370}
SPL {X  -156.829, Y  +350.854, Z    +0.000, E1   -20.141, E3 -300793.923}
SPL {X  -159.049, Y  +365.169, Z    +0.000, E1   -12.580, E3 -300798.667}
SPL {X  -159.776, Y  +374.231, Z    +0.000, E1    -7.281, E3 -300800.553}
SPL {X  -159.986, Y  +381.380, Z    +0.000, E1    -2.685, E3 -300801.399}
SPL {X  -159.990, Y  +384.493, Z    +0.000, E1    -0.324, E3 -300801.607}
SPL {X  -159.990, Y  +387.327, Z    +0.000, E1    +2.137, E3 -300801.790}
SPL {X  -159.990, Y  +392.053, Z    +0.000, E1    +7.477, E3 -300802.255}
SPL {X  -159.990, Y  +396.158, Z    +0.000, E1   +12.775, E3 -300802.881}
SPL {X  -159.990, Y  +401.377, Z    +0.000, E1   +19.398, E3 -300804.061}
SPL {X  -159.990, Y  +411.365, Z    +0.000, E1   +30.630, E3 -300807.269}
SPL {X  -159.990, Y  +450.467, Z    +0.000, E1   +50.183, E3 -300830.918}
SPL {X  -159.990, Y  +509.934, Z    +0.000, E1   +54.923, E3 -300893.537}
SPL {X  -159.990, Y  +516.848, Z    +0.000, E1   +54.930, E3 -300903.825}
SPL {X  -159.990, Y  +524.818, Z    +0.000, E1   +54.933, E3 -300915.697}
SPL {X  -159.990, Y  +532.100, Z    +0.000, E1   +54.924, E3 -300926.550}
SPL {X  -159.990, Y  +539.391, Z    +0.000, E1   +54.933, E3 -300937.402}
SPL {X  -159.990, Y  +546.283, Z    +0.000, E1   +54.924, E3 -300947.674}
SPL {X  -159.990, Y  +553.734, Z    +0.000, E1   +54.938, E3 -300958.760}
SPL {X  -159.990, Y  +564.956, Z    +0.000, E1   +54.973, E3 -300975.432}
SPL {X  -159.990, Y  +575.140, Z    +0.000, E1   +54.928, E3 -300990.665}
SPL {X  -159.990, Y  +581.046, Z    +0.000, E1   +54.920, E3 -300999.477}
SPL {X  -159.990, Y  +588.063, Z    +0.000, E1   +54.931, E3 -301009.912}
SPL {X  -159.990, Y  +595.273, Z    +0.000, E1   +54.928, E3 -301020.636}
SPL {X  -159.990, Y  +602.326, Z    +0.000, E1   +54.932, E3 -301031.136}
SPL {X  -159.990, Y  +610.296, Z    +0.000, E1   +54.937, E3 -301043.006}
SPL {X  -159.990, Y  +618.534, Z    +0.000, E1   +54.942, E3 -301055.243}
SPL {X  -159.990, Y  +625.928, Z    +0.000, E1   +54.931, E3 -301066.268}
SPL {X  -159.990, Y  +633.423, Z    +0.000, E1   +54.943, E3 -301077.410}
SPL {X  -159.990, Y  +640.333, Z    +0.000, E1   +54.927, E3 -301087.724}
SPL {X  -159.990, Y  +648.272, Z    +0.000, E1   +54.961, E3 -301099.472}
SPL {X  -159.990, Y  +655.990, Z    +0.000, E1   +54.930, E3 -301111.019}
SPL {X  -159.990, Y  +665.734, Z    +0.000, E1   +54.984, E3 -301125.470}
SPL {X  -159.953, Y  +674.920, Z    +0.000, E1   +54.918, E3 -301139.282}
SPL {X  -159.714, Y  +680.893, Z    +0.000, E1   +54.890, E3 -301148.422}
SPL {X  -159.222, Y  +687.156, Z    +0.000, E1   +54.792, E3 -301158.309}
SPL {X  -158.388, Y  +694.082, Z    +0.000, E1   +54.679, E3 -301169.447}
SPL {X  -157.277, Y  +700.838, Z    +0.000, E1   +54.465, E3 -301180.704}
SPL {X  -156.153, Y  +706.327, Z    +0.000, E1   +54.274, E3 -301190.040}
SPL {X  -154.917, Y  +711.470, Z    +0.000, E1   +54.052, E3 -301198.991}
SPL {X  -153.204, Y  +717.603, Z    +0.000, E1   +53.775, E3 -301209.838}
SPL {X  -151.355, Y  +723.351, Z    +0.000, E1   +53.415, E3 -301220.309}
SPL {X  -149.371, Y  +728.816, Z    +0.000, E1   +53.074, E3 -301230.400}
SPL {X  -147.376, Y  +733.767, Z    +0.000, E1   +52.671, E3 -301239.802}
SPL {X  -145.158, Y  +738.775, Z    +0.000, E1   +52.288, E3 -301249.353}
SPL {X  -142.385, Y  +744.461, Z    +0.000, E1   +51.729, E3 -301260.465}
SPL {X  -132.301, Y  +761.463, Z    +0.000, E1   +45.510, E3 -301338.203}
ENDSPLINE

SPLINE
SPL {X  -145.877, Y  +737.201, Z    +0.000, E1   +34.468, E3 -301421.314}
SPL {X  -152.550, Y  +719.721, Z    +0.000, E1   +27.728, E3 -301436.804}
SPL {X  -157.145, Y  +701.536, Z    +0.000, E1   +19.368, E3 -301446.258}
SPL {X  -159.035, Y  +688.952, Z    +0.000, E1   +12.676, E3 -301450.299}
SPL {X  -159.756, Y  +680.154, Z    +0.000, E1    +7.520, E3 -301452.026}
SPL {X  -159.986, Y  +672.560, Z    +0.000, E1    +2.636, E3 -301452.924}
SPL {X  -159.990, Y  +669.364, Z    +0.000, E1    +0.170, E3 -301453.131}
SPL {X  -159.990, Y  +666.603, Z    +0.000, E1    -2.256, E3 -301453.303}
SPL {X  -159.990, Y  +662.759, Z    +0.000, E1    -6.725, E3 -301453.646}
SPL {X  -159.990, Y  +658.737, Z    +0.000, E1   -11.801, E3 -301454.224}
SPL {X  -159.990, Y  +652.023, Z    +0.000, E1   -20.449, E3 -301455.709}
SPL {X  -159.990, Y  +641.935, Z    +0.000, E1   -31.848, E3 -301458.881}
SPL {X  -159.990, Y  +605.095, Z    +0.000, E1   -49.514, E3 -301483.087}
SPL {X  -159.990, Y  +543.998, Z    +0.000, E1   -54.483, E3 -301549.077}
SPL {X  -159.990, Y  +535.878, Z    +0.000, E1   -54.465, E3 -301561.412}
SPL {X  -159.990, Y  +529.394, Z    +0.000, E1   -54.464, E3 -301571.241}
SPL {X  -159.990, Y  +521.536, Z    +0.000, E1   -54.480, E3 -301583.123}
SPL {X  -159.990, Y  +514.089, Z    +0.000, E1   -54.461, E3 -301594.435}
SPL {X  -159.990, Y  +506.373, Z    +0.000, E1   -54.484, E3 -301606.072}
SPL {X  -159.990, Y  +497.571, Z    +0.000, E1   -54.478, E3 -301619.415}
SPL {X  -159.990, Y  +490.343, Z    +0.000, E1   -54.468, E3 -301630.380}
SPL {X  -159.990, Y  +483.191, Z    +0.000, E1   -54.478, E3 -301641.196}
SPL {X  -159.990, Y  +475.502, Z    +0.000, E1   -54.476, E3 -301652.845}
SPL {X  -159.990, Y  +448.520, Z    +0.000, E1   -58.543, E3 -301664.474}
SPL {X  -159.990, Y  +438.044, Z    +0.000, E1   -58.687, E3 -301677.111}
SPL {X  -159.990, Y  +431.936, Z    +0.000, E1   -57.955, E3 -301689.931}
SPL {X  -159.990, Y  +427.860, Z    +0.000, E1   -57.091, E3 -301700.994}
SPL {X  -159.990, Y  +424.653, Z    +0.000, E1   -55.901, E3 -301713.300}
SPL {X  -159.990, Y  +419.503, Z    +0.000, E1   -55.092, E3 -301725.825}
ENDSPLINE

SPLINE
SPL {X  -159.990, Y  +431.130, Z    +0.000, E1   -50.080, E3 -301738.200}
ENDSPLINE

SPLINE
SPL {X  -159.990, Y  +421.718, Z    +0.000, E1   -50.072, E3 -301754.965}
SPL {X  -159.990, Y  +412.896, Z    +0.000, E1   -50.065, E3 -301770.658}
SPL {X  -159.990, Y  +403.654, Z    +0.000, E1   -50.076, E3 -301787.065}
SPL {X  -159.990, Y  +394.612, Z    +0.000, E1   -50.064, E3 -301803.153}
SPL {X  -159.990, Y  +387.356, Z    +0.000, E1   -50.042, E3 -301816.100}
SPL {X  -159.956, Y  +379.183, Z    +0.000, E1   -50.071, E3 -301830.614}
SPL {X  -159.545, Y  +370.569, Z    +0.000, E1   -49.982, E3 -301846.380}
SPL {X  -158.871, Y  +363.614, Z    +0.000, E1   -49.855, E3 -301859.459}
SPL {X  -158.179, Y  +358.495, Z    +0.000, E1   -49.715, E3 -301869.308}
SPL {X  -157.354, Y  +353.576, Z    +0.000, E1   -49.583, E3 -301878.894}
SPL {X  -156.029, Y  +347.121, Z    +0.000, E1   -49.358, E3 -301891.711}
SPL {X  -154.686, Y  +341.646, Z    +0.000, E1   -49.094, E3 -301902.855}
SPL {X  -153.089, Y  +336.017, Z    +0.000, E1   -48.817, E3 -301914.464}
SPL {X  -151.481, Y  +331.019, Z    +0.000, E1   -48.491, E3 -301925.012}
SPL {X  -149.787, Y  +326.281, Z    +0.000, E1   -48.192, E3 -301935.100}
SPL {X  -147.422, Y  +320.342, Z    +0.000, E1   -47.750, E3 -301947.968}
SPL {X  -145.797, Y  +316.621, Z    +0.000, E1   -47.387, E3 -301956.210}
SPL {X  -141.189, Y  +307.250, Z    +0.000, E1   -40.067, E3 -302038.810}
ENDSPLINE

SPLINE
SPL {X  -154.923, Y  +342.556, Z    +0.000, E1   -23.930, E3 -302100.309}
SPL {X  -158.138, Y  +358.230, Z    +0.000, E1   -16.243, E3 -302109.267}
SPL {X  -159.647, Y  +372.034, Z    +0.000, E1    -8.739, E3 -302113.631}
SPL {X  -159.989, Y  +381.927, Z    +0.000, E1    -2.565, E3 -302115.391}
SPL {X  -159.990, Y  +386.909, Z    +0.000, E1    +1.211, E3 -302115.934}
SPL {X  -159.990, Y  +390.921, Z    +0.000, E1    +5.111, E3 -302116.413}
SPL {X  -159.990, Y  +395.719, Z    +0.000, E1   +10.396, E3 -302117.232}
SPL {X  -159.990, Y  +400.739, Z    +0.000, E1   +16.236, E3 -302118.430}
SPL {X  -159.990, Y  +409.482, Z    +0.000, E1   +25.418, E3 -302121.635}
SPL {X  -159.990, Y  +440.741, Z    +0.000, E1   +43.570, E3 -302142.292}
SPL {X  -159.990, Y  +488.072, Z    +0.000, E1   +48.834, E3 -302203.414}
SPL {X  -159.990, Y  +495.397, Z    +0.000, E1   +48.860, E3 -302216.963}
SPL {X  -159.990, Y  +502.531, Z    +0.000, E1   +48.834, E3 -302230.242}
SPL {X  -159.990, Y  +508.013, Z    +0.000, E1   +48.835, E3 -302240.377}
SPL {X  -159.990, Y  +513.813, Z    +0.000, E1   +48.843, E3 -302251.125}
SPL {X  -159.990, Y  +522.177, Z    +0.000, E1   +48.881, E3 -302266.602}
SPL {X  -159.990, Y  +532.076, Z    +0.000, E1   +48.872, E3 -302284.975}
SPL {X  -159.990, Y  +539.248, Z    +0.000, E1   +48.832, E3 -302298.343}
SPL {X  -159.990, Y  +544.926, Z    +0.000, E1   +48.835, E3 -302308.872}
SPL {X  -159.990, Y  +550.252, Z    +0.000, E1   +48.827, E3 -302318.778}
SPL {X  -159.990, Y  +555.692, Z    +0.000, E1   +48.830, E3 -302328.875}
SPL {X  -159.990, Y  +561.308, Z    +0.000, E1   +48.827, E3 -302339.322}
SPL {X  -159.990, Y  +566.669, Z    +0.000, E1   +48.820, E3 -302349.271}
SPL {X  -159.990, Y  +572.248, Z    +0.000, E1   +48.830, E3 -302359.616}
SPL {X  -159.990, Y  +577.770, Z    +0.000, E1   +48.821, E3 -302369.863}
SPL {X  -159.990, Y  +583.108, Z    +0.000, E1   +48.828, E3 -302379.765}
SPL {X  -159.990, Y  +588.804, Z    +0.000, E1   +48.829, E3 -302390.322}
SPL {X  -159.990, Y  +594.280, Z    +0.000, E1   +48.826, E3 -302400.484}
SPL {X  -159.990, Y  +600.107, Z    +0.000, E1   +48.833, E3 -302411.298}
SPL {X  -159.990, Y  +605.910, Z    +0.000, E1   +48.823, E3 -302422.077}
SPL {X  -159.990, Y  +611.566, Z    +0.000, E1   +48.829, E3 -302432.566}
SPL {X  -159.990, Y  +617.357, Z    +0.000, E1   +48.824, E3 -302443.321}
SPL {X  -159.990, Y  +622.965, Z    +0.000, E1   +48.826, E3 -302453.720}
SPL {X  -159.990, Y  +629.255, Z    +0.000, E1   +48.834, E3 -302465.387}
SPL {X  -159.990, Y  +634.905, Z    +0.000, E1   +48.821, E3 -302475.884}
SPL {X  -159.990, Y  +640.372, Z    +0.000, E1   +48.828, E3 -302486.021}
SPL {X  -159.990, Y  +646.939, Z    +0.000, E1   +48.838, E3 -302498.191}
SPL {X  -159.990, Y  +653.448, Z    +0.000, E1   +48.827, E3 -302510.286}
SPL {X  -159.990, Y  +659.039, Z    +0.000, E1   +48.826, E3 -302520.650}
SPL {X  -159.990, Y  +664.817, Z    +0.000, E1   +48.832, E3 -302531.365}
SPL {X  -159.990, Y  +671.221, Z    +0.000, E1   +48.836, E3 -302543.238}
SPL {X  -159.887, Y  +677.230, Z    +0.000, E1   +48.811, E3 -302554.504}
SPL {X  -159.602, Y  +682.629, Z    +0.000, E1   +48.761, E3 -302564.837}
SPL {X  -159.150, Y  +687.876, Z    +0.000, E1   +48.673, E3 -302575.076}
SPL {X  -158.569, Y  +692.776, Z    +0.000, E1   +48.570, E3 -302584.784}
SPL {X  -157.870, Y  +697.458, Z    +0.000, E1   +48.439, E3 -302594.213}
SPL {X  -157.028, Y  +702.144, Z    +0.000, E1   +48.297, E3 -302603.761}
SPL {X  -155.977, Y  +707.110, Z    +0.000, E1   +48.106, E3 -302614.065}
SPL {X  -154.657, Y  +712.464, Z    +0.000, E1   +47.874, E3 -302625.349}
SPL {X  -153.406, Y  +716.924, Z    +0.000, E1   +47.628, E3 -302634.915}
SPL {X  -152.020, Y  +721.367, Z    +0.000, E1   +47.374, E3 -302644.566}
SPL {X  -150.440, Y  +725.947, Z    +0.000, E1   +47.070, E3 -302654.671}
SPL {X  -148.730, Y  +730.459, Z    +0.000, E1   +46.749, E3 -302664.722}
SPL {X  -147.178, Y  +734.233, Z    +0.000, E1   +46.439, E3 -302673.256}
SPL {X  -140.222, Y  +748.536, Z    +0.000, E1   +42.074, E3 -302738.232}
ENDSPLINE

SPLINE
SPL {X  -152.021, Y  +721.365, Z    +0.000, E1   +28.339, E3 -302813.623}
SPL {X  -158.165, Y  +695.595, Z    +0.000, E1   +16.189, E3 -302830.706}
SPL {X  -159.572, Y  +683.063, Z    +0.000, E1    +9.282, E3 -302834.713}
SPL {X  -159.928, Y  +675.946, Z    +0.000, E1    +5.007, E3 -302836.134}
SPL {X  -159.990, Y  +669.697, Z    +0.000, E1    +0.851, E3 -302836.894}
SPL {X  -159.990, Y  +665.698, Z    +0.000, E1    -2.616, E3 -302837.273}
SPL {X  -159.990, Y  +662.251, Z    +0.000, E1    -6.155, E3 -302837.719}
SPL {X  -159.990, Y  +658.551, Z    +0.000, E1   -10.313, E3 -302838.371}
SPL {X  -159.990, Y  +653.526, Z    +0.000, E1   -16.156, E3 -302839.606}
SPL {X  -159.990, Y  +644.434, Z    +0.000, E1   -25.921, E3 -302842.801}
SPL {X  -159.990, Y  +612.255, Z    +0.000, E1   -44.102, E3 -302864.682}
SPL {X  -159.990, Y  +561.053, Z    +0.000, E1   -49.668, E3 -302929.515}
SPL {X  -159.990, Y  +552.984, Z    +0.000, E1   -49.619, E3 -302944.156}
SPL {X  -159.990, Y  +547.278, Z    +0.000, E1   -49.619, E3 -302954.455}
SPL {X  -159.990, Y  +538.738, Z    +0.000, E1   -49.672, E3 -302969.779}
SPL {X  -159.990, Y  +529.436, Z    +0.000, E1   -49.638, E3 -302986.603}
SPL {X  -159.990, Y  +522.804, Z    +0.000, E1   -49.620, E3 -302998.592}
SPL {X  -159.990, Y  +515.173, Z    +0.000, E1   -49.653, E3 -303012.330}
SPL {X  -159.990, Y  +505.472, Z    +0.000, E1   -49.465, E3 -303031.135}
ENDSPLINE

SPLINE
SPL {X  -159.990, Y  +518.841, Z    +0.000, E1   -41.643, E3 -303049.543}
ENDSPLINE

SPLINE
SPL {X  -159.990, Y  +508.096, Z    +0.000, E1   -42.952, E3 -303066.810}
SPL {X  -159.990, Y  +500.642, Z    +0.000, E1   -43.747, E3 -303078.731}
SPL {X  -159.990, Y  +495.820, Z    +0.000, E1   -44.207, E3 -303086.618}
SPL {X  -159.990, Y  +487.435, Z    +0.000, E1   -45.185, E3 -303098.910}
SPL {X  -159.990, Y  +477.648, Z    +0.000, E1   -46.080, E3 -303113.907}
SPL {X  -159.990, Y  +469.952, Z    +0.000, E1   -46.750, E3 -303125.415}
SPL {X  -159.990, Y  +462.892, Z    +0.000, E1   -47.497, E3 -303134.899}
SPL {X  -159.990, Y  +452.841, Z    +0.000, E1   -48.572, E3 -303147.746}
SPL {X  -159.990, Y  +439.038, Z    +0.000, E1   -49.804, E3 -303165.798}
SPL {X  -159.990, Y  +429.517, Z    +0.000, E1   -50.043, E3 -303181.146}
SPL {X  -159.990, Y  +423.834, Z    +0.000, E1   -50.037, E3 -303191.258}
SPL {X  -159.990, Y  +417.693, Z    +0.000, E1   -50.049, E3 -303202.156}
SPL {X  -159.990, Y  +411.447, Z    +0.000, E1   -50.039, E3 -303213.275}
SPL {X  -159.990, Y  +406.170, Z    +0.000, E1   -50.036, E3 -303222.647}
SPL {X  -159.990, Y  +399.787, Z    +0.000, E1   -50.064, E3 -303233.955}
SPL {X  -159.990, Y  +393.038, Z    +0.000, E1   -50.038, E3 -303245.989}
SPL {X  -159.990, Y  +387.356, Z    +0.000, E1   -50.042, E3 -303256.100}
SPL {X  -159.990, Y  +382.225, Z    +0.000, E1   -50.028, E3 -303265.245}
SPL {X  -159.846, Y  +375.718, Z    +0.000, E1   -50.041, E3 -303276.901}
SPL {X  -159.443, Y  +369.277, Z    +0.000, E1   -49.941, E3 -303288.815}
SPL {X  -158.871, Y  +363.614, Z    +0.000, E1   -49.855, E3 -303299.459}
SPL {X  -158.179, Y  +358.495, Z    +0.000, E1   -49.715, E3 -303309.308}
SPL {X  -157.077, Y  +352.107, Z    +0.000, E1   -49.567, E3 -303321.742}
SPL {X  -155.744, Y  +345.884, Z    +0.000, E1   -49.283, E3 -303334.229}
SPL {X  -154.686, Y  +341.646, Z    +0.000, E1   -49.094, E3 -303342.855}
SPL {X  -153.439, Y  +337.188, Z    +0.000, E1   -48.857, E3 -303352.062}
SPL {X  -151.836, Y  +332.074, Z    +0.000, E1   -48.585, E3 -303362.738}
SPL {X  -150.221, Y  +327.451, Z    +0.000, E1   -48.251, E3 -303372.616}
SPL {X  -148.587, Y  +323.181, Z    +0.000, E1   -47.960, E3 -303381.800}
SPL {X  -146.510, Y  +318.222, Z    +0.000, E1   -47.558, E3 -303392.636}
SPL {X  -141.189, Y  +307.250, Z    +0.000, E1   -40.067, E3 -303478.810}
ENDSPLINE

SPLINE
SPL {X  -154.923, Y  +342.556, Z    +0.000, E1   -23.930, E3 -303540.309}
SPL {X  -158.138, Y  +358.230, Z    +0.000, E1   -16.243, E3 -303549.267}
SPL {X  -159.647, Y  +372.034, Z    +0.000, E1    -8.739, E3 -303553.631}
SPL {X  -159.989, Y  +381.927, Z    +0.000, E1    -2.565, E3 -303555.391}
SPL {X  -159.990, Y  +386.909, Z    +0.000, E1    +1.211, E3 -303555.934}
SPL {X  -159.990, Y  +390.921, Z    +0.000, E1    +5.111, E3 -303556.413}
SPL {X  -159.990, Y  +395.719, Z    +0.000, E1   +10.396, E3 -303557.232}
SPL {X  -159.990, Y  +400.739, Z    +0.000, E1   +16.236, E3 -303558.430}
SPL {X  -159.990, Y  +409.482, Z    +0.000, E1   +25.418, E3 -303561.635}
SPL {X  -159.990, Y  +440.741, Z    +0.000, E1   +43.570, E3 -303582.292}
SPL {X  -159.990, Y  +489.732, Z    +0.000, E1   +48.863, E3 -303646.450}
SPL {X  -159.990, Y  +496.901, Z    +0.000, E1   +48.832, E3 -303659.797}
SPL {X  -159.990, Y  +502.531, Z    +0.000, E1   +48.834, E3 -303670.242}
SPL {X  -159.990, Y  +508.013, Z    +0.000, E1   +48.835, E3 -303680.377}
SPL {X  -159.990, Y  +513.813, Z    +0.000, E1   +48.843, E3 -303691.125}
SPL {X  -159.990, Y  +522.177, Z    +0.000, E1   +48.881, E3 -303706.602}
SPL {X  -159.990, Y  +532.076, Z    +0.000, E1   +48.872, E3 -303724.975}
SPL {X  -159.990, Y  +539.248, Z    +0.000, E1   +48.832, E3 -303738.343}
SPL {X  -159.990, Y  +544.926, Z    +0.000, E1   +48.835, E3 -303748.872}
SPL {X  -159.990, Y  +550.252, Z    +0.000, E1   +48.827, E3 -303758.778}
SPL {X  -159.990, Y  +555.692, Z    +0.000, E1   +48.830, E3 -303768.875}
SPL {X  -159.990, Y  +561.308, Z    +0.000, E1   +48.827, E3 -303779.322}
SPL {X  -159.990, Y  +566.669, Z    +0.000, E1   +48.820, E3 -303789.271}
SPL {X  -159.990, Y  +572.248, Z    +0.000, E1   +48.830, E3 -303799.616}
SPL {X  -159.990, Y  +577.770, Z    +0.000, E1   +48.821, E3 -303809.863}
SPL {X  -159.990, Y  +583.108, Z    +0.000, E1   +48.828, E3 -303819.765}
SPL {X  -159.990, Y  +588.804, Z    +0.000, E1   +48.829, E3 -303830.322}
SPL {X  -159.990, Y  +594.280, Z    +0.000, E1   +48.826, E3 -303840.484}
SPL {X  -159.990, Y  +600.107, Z    +0.000, E1   +48.833, E3 -303851.298}
SPL {X  -159.990, Y  +605.910, Z    +0.000, E1   +48.823, E3 -303862.077}
SPL {X  -159.990, Y  +611.566, Z    +0.000, E1   +48.829, E3 -303872.566}
SPL {X  -159.990, Y  +617.357, Z    +0.000, E1   +48.824, E3 -303883.321}
SPL {X  -159.990, Y  +622.965, Z    +0.000, E1   +48.826, E3 -303893.720}
SPL {X  -159.990, Y  +629.255, Z    +0.000, E1   +48.834, E3 -303905.387}
SPL {X  -159.990, Y  +634.905, Z    +0.000, E1   +48.821, E3 -303915.884}
SPL {X  -159.990, Y  +640.372, Z    +0.000, E1   +48.828, E3 -303926.021}
SPL {X  -159.990, Y  +646.939, Z    +0.000, E1   +48.838, E3 -303938.191}
SPL {X  -159.990, Y  +653.448, Z    +0.000, E1   +48.827, E3 -303950.286}
SPL {X  -159.990, Y  +659.039, Z    +0.000, E1   +48.826, E3 -303960.650}
SPL {X  -159.990, Y  +664.817, Z    +0.000, E1   +48.832, E3 -303971.365}
SPL {X  -159.990, Y  +671.221, Z    +0.000, E1   +48.836, E3 -303983.238}
SPL {X  -159.887, Y  +677.230, Z    +0.000, E1   +48.811, E3 -303994.504}
SPL {X  -159.602, Y  +682.629, Z    +0.000, E1   +48.761, E3 -304004.837}
SPL {X  -159.150, Y  +687.876, Z    +0.000, E1   +48.673, E3 -304015.076}
SPL {X  -158.569, Y  +692.776, Z    +0.000, E1   +48.570, E3 -304024.784}
SPL {X  -157.870, Y  +697.458, Z    +0.000, E1   +48.439, E3 -304034.213}
SPL {X  -157.028, Y  +702.144, Z    +0.000, E1   +48.297, E3 -304043.761}
SPL {X  -155.977, Y  +707.110, Z    +0.000, E1   +48.106, E3 -304054.065}
SPL {X  -154.657, Y  +712.464, Z    +0.000, E1   +47.874, E3 -304065.349}
SPL {X  -153.406, Y  +716.924, Z    +0.000, E1   +47.628, E3 -304074.915}
SPL {X  -152.020, Y  +721.367, Z    +0.000, E1   +47.374, E3 -304084.566}
SPL {X  -150.440, Y  +725.947, Z    +0.000, E1   +47.070, E3 -304094.671}
SPL {X  -148.730, Y  +730.459, Z    +0.000, E1   +46.749, E3 -304104.722}
SPL {X  -147.178, Y  +734.233, Z    +0.000, E1   +46.439, E3 -304113.256}
SPL {X  -140.263, Y  +748.461, Z    +0.000, E1   +42.675, E3 -304171.594}
ENDSPLINE

SPLINE
SPL {X  -141.835, Y  +745.525, Z    +0.000, E1   +39.068, E3 -304203.595}
SPL {X  -152.406, Y  +720.176, Z    +0.000, E1   +27.814, E3 -304254.808}
SPL {X  -158.165, Y  +695.595, Z    +0.000, E1   +16.189, E3 -304270.706}
SPL {X  -159.572, Y  +683.063, Z    +0.000, E1    +9.282, E3 -304274.713}
SPL {X  -159.928, Y  +675.946, Z    +0.000, E1    +5.007, E3 -304276.134}
SPL {X  -159.990, Y  +671.468, Z    +0.000, E1    +2.030, E3 -304276.730}
SPL {X  -159.990, Y  +667.678, Z    +0.000, E1    -0.783, E3 -304277.080}
SPL {X  -159.990, Y  +663.139, Z    +0.000, E1    -5.135, E3 -304277.597}
SPL {X  -159.990, Y  +658.551, Z    +0.000, E1   -10.313, E3 -304278.371}
SPL {X  -159.990, Y  +653.526, Z    +0.000, E1   -16.156, E3 -304279.606}
SPL {X  -159.990, Y  +644.434, Z    +0.000, E1   -25.921, E3 -304282.801}
SPL {X  -159.990, Y  +612.255, Z    +0.000, E1   -44.102, E3 -304304.682}
SPL {X  -159.990, Y  +561.053, Z    +0.000, E1   -49.668, E3 -304369.515}
SPL {X  -159.990, Y  +552.984, Z    +0.000, E1   -49.619, E3 -304384.156}
SPL {X  -159.990, Y  +547.278, Z    +0.000, E1   -49.619, E3 -304394.455}
SPL {X  -159.990, Y  +538.738, Z    +0.000, E1   -49.672, E3 -304409.779}
SPL {X  -159.990, Y  +529.436, Z    +0.000, E1   -49.638, E3 -304426.603}
SPL {X  -159.990, Y  +522.804, Z    +0.000, E1   -49.620, E3 -304438.592}
SPL {X  -159.990, Y  +515.173, Z    +0.000, E1   -49.653, E3 -304452.330}
SPL {X  -159.990, Y  +505.472, Z    +0.000, E1   -49.465, E3 -304471.135}
ENDSPLINE

SPLINE
SPL {X  -159.990, Y  +520.622, Z    +0.000, E1   -41.395, E3 -304486.672}
ENDSPLINE

SPLINE
SPL {X  -159.990, Y  +512.735, Z    +0.000, E1   -42.369, E3 -304499.523}
SPL {X  -159.990, Y  +505.924, Z    +0.000, E1   -43.199, E3 -304510.181}
SPL {X  -159.990, Y  +497.983, Z    +0.000, E1   -44.027, E3 -304523.054}
SPL {X  -159.990, Y  +489.703, Z    +0.000, E1   -44.938, E3 -304535.473}
SPL {X  -159.990, Y  +484.712, Z    +0.000, E1   -45.426, E3 -304543.087}
SPL {X  -159.990, Y  +477.648, Z    +0.000, E1   -46.080, E3 -304553.907}
SPL {X  -159.990, Y  +469.952, Z    +0.000, E1   -46.750, E3 -304565.415}
SPL {X  -159.990, Y  +462.892, Z    +0.000, E1   -47.497, E3 -304574.899}
SPL {X  -159.990, Y  +452.841, Z    +0.000, E1   -48.572, E3 -304587.746}
SPL {X  -159.990, Y  +439.038, Z    +0.000, E1   -49.804, E3 -304605.798}
SPL {X  -159.990, Y  +429.517, Z    +0.000, E1   -50.043, E3 -304621.146}
SPL {X  -159.990, Y  +423.834, Z    +0.000, E1   -50.037, E3 -304631.258}
SPL {X  -159.990, Y  +417.693, Z    +0.000, E1   -50.049, E3 -304642.156}
SPL {X  -159.990, Y  +411.447, Z    +0.000, E1   -50.039, E3 -304653.275}
SPL {X  -159.990, Y  +406.170, Z    +0.000, E1   -50.036, E3 -304662.647}
SPL {X  -159.990, Y  +399.787, Z    +0.000, E1   -50.064, E3 -304673.955}
SPL {X  -159.990, Y  +393.038, Z    +0.000, E1   -50.038, E3 -304685.989}
SPL {X  -159.990, Y  +387.356, Z    +0.000, E1   -50.042, E3 -304696.100}
SPL {X  -159.956, Y  +379.183, Z    +0.000, E1   -50.071, E3 -304710.614}
SPL {X  -159.413, Y  +368.921, Z    +0.000, E1   -49.998, E3 -304729.389}
SPL {X  -158.412, Y  +360.086, Z    +0.000, E1   -49.787, E3 -304746.191}
SPL {X  -157.354, Y  +353.576, Z    +0.000, E1   -49.583, E3 -304758.894}
SPL {X  -156.029, Y  +347.121, Z    +0.000, E1   -49.358, E3 -304771.711}
SPL {X  -154.686, Y  +341.646, Z    +0.000, E1   -49.094, E3 -304782.855}
SPL {X  -153.439, Y  +337.188, Z    +0.000, E1   -48.857, E3 -304792.062}
SPL {X  -151.836, Y  +332.074, Z    +0.000, E1   -48.585, E3 -304802.738}
SPL {X  -149.787, Y  +326.281, Z    +0.000, E1   -48.192, E3 -304815.100}
SPL {X  -148.124, Y  +322.035, Z    +0.000, E1   -47.846, E3 -304824.324}
SPL {X  -146.510, Y  +318.222, Z    +0.000, E1   -47.558, E3 -304832.636}
SPL {X  -141.189, Y  +307.250, Z    +0.000, E1   -40.067, E3 -304918.810}
ENDSPLINE

SPLINE
SPL {X  -154.923, Y  +342.556, Z    +0.000, E1   -23.930, E3 -304980.309}
SPL {X  -158.138, Y  +358.230, Z    +0.000, E1   -16.243, E3 -304989.267}
SPL {X  -159.647, Y  +372.034, Z    +0.000, E1    -8.739, E3 -304993.631}
SPL {X  -159.969, Y  +379.932, Z    +0.000, E1    -3.817, E3 -304995.139}
SPL {X  -159.990, Y  +384.616, Z    +0.000, E1    -0.627, E3 -304995.691}
SPL {X  -159.990, Y  +387.962, Z    +0.000, E1    +2.241, E3 -304996.048}
SPL {X  -159.990, Y  +390.921, Z    +0.000, E1    +5.111, E3 -304996.413}
SPL {X  -159.990, Y  +395.719, Z    +0.000, E1   +10.396, E3 -304997.232}
SPL {X  -159.990, Y  +400.739, Z    +0.000, E1   +16.236, E3 -304998.430}
SPL {X  -159.990, Y  +409.482, Z    +0.000, E1   +25.418, E3 -305001.635}
SPL {X  -159.990, Y  +440.741, Z    +0.000, E1   +43.570, E3 -305022.292}
SPL {X  -159.990, Y  +489.732, Z    +0.000, E1   +48.863, E3 -305086.450}
SPL {X  -159.990, Y  +496.901, Z    +0.000, E1   +48.832, E3 -305099.797}
SPL {X  -159.990, Y  +502.531, Z    +0.000, E1   +48.834, E3 -305110.242}
SPL {X  -159.990, Y  +508.013, Z    +0.000, E1   +48.835, E3 -305120.377}
SPL {X  -159.990, Y  +513.813, Z    +0.000, E1   +48.843, E3 -305131.125}
SPL {X  -159.990, Y  +522.177, Z    +0.000, E1   +48.881, E3 -305146.602}
SPL {X  -159.990, Y  +532.076, Z    +0.000, E1   +48.872, E3 -305164.975}
SPL {X  -159.990, Y  +539.248, Z    +0.000, E1   +48.832, E3 -305178.343}
SPL {X  -159.990, Y  +544.926, Z    +0.000, E1   +48.835, E3 -305188.872}
SPL {X  -159.990, Y  +550.252, Z    +0.000, E1   +48.827, E3 -305198.778}
SPL {X  -159.990, Y  +555.692, Z    +0.000, E1   +48.830, E3 -305208.875}
SPL {X  -159.990, Y  +561.308, Z    +0.000, E1   +48.827, E3 -305219.322}
SPL {X  -159.990, Y  +566.669, Z    +0.000, E1   +48.820, E3 -305229.271}
SPL {X  -159.990, Y  +572.248, Z    +0.000, E1   +48.830, E3 -305239.616}
SPL {X  -159.990, Y  +577.770, Z    +0.000, E1   +48.821, E3 -305249.863}
SPL {X  -159.990, Y  +583.108, Z    +0.000, E1   +48.828, E3 -305259.765}
SPL {X  -159.990, Y  +588.804, Z    +0.000, E1   +48.829, E3 -305270.322}
SPL {X  -159.990, Y  +594.280, Z    +0.000, E1   +48.826, E3 -305280.484}
SPL {X  -159.990, Y  +600.107, Z    +0.000, E1   +48.833, E3 -305291.298}
SPL {X  -159.990, Y  +605.910, Z    +0.000, E1   +48.823, E3 -305302.077}
SPL {X  -159.990, Y  +611.566, Z    +0.000, E1   +48.829, E3 -305312.566}
SPL {X  -159.990, Y  +617.357, Z    +0.000, E1   +48.824, E3 -305323.321}
SPL {X  -159.990, Y  +622.965, Z    +0.000, E1   +48.826, E3 -305333.720}
SPL {X  -159.990, Y  +629.255, Z    +0.000, E1   +48.834, E3 -305345.387}
SPL {X  -159.990, Y  +634.905, Z    +0.000, E1   +48.821, E3 -305355.884}
SPL {X  -159.990, Y  +640.372, Z    +0.000, E1   +48.828, E3 -305366.021}
SPL {X  -159.990, Y  +646.939, Z    +0.000, E1   +48.838, E3 -305378.191}
SPL {X  -159.990, Y  +653.448, Z    +0.000, E1   +48.827, E3 -305390.286}
SPL {X  -159.990, Y  +659.039, Z    +0.000, E1   +48.826, E3 -305400.650}
SPL {X  -159.990, Y  +664.817, Z    +0.000, E1   +48.832, E3 -305411.365}
SPL {X  -159.990, Y  +671.221, Z    +0.000, E1   +48.836, E3 -305423.238}
SPL {X  -159.887, Y  +677.230, Z    +0.000, E1   +48.811, E3 -305434.504}
SPL {X  -159.602, Y  +682.629, Z    +0.000, E1   +48.761, E3 -305444.837}
SPL {X  -159.150, Y  +687.876, Z    +0.000, E1   +48.673, E3 -305455.076}
SPL {X  -158.569, Y  +692.776, Z    +0.000, E1   +48.570, E3 -305464.784}
SPL {X  -157.870, Y  +697.458, Z    +0.000, E1   +48.439, E3 -305474.213}
SPL {X  -157.028, Y  +702.144, Z    +0.000, E1   +48.297, E3 -305483.761}
SPL {X  -155.977, Y  +707.110, Z    +0.000, E1   +48.106, E3 -305494.065}
SPL {X  -154.657, Y  +712.464, Z    +0.000, E1   +47.874, E3 -305505.349}
SPL {X  -153.406, Y  +716.924, Z    +0.000, E1   +47.628, E3 -305514.915}
SPL {X  -152.020, Y  +721.367, Z    +0.000, E1   +47.374, E3 -305524.566}
SPL {X  -150.440, Y  +725.947, Z    +0.000, E1   +47.070, E3 -305534.671}
SPL {X  -148.730, Y  +730.459, Z    +0.000, E1   +46.749, E3 -305544.722}
SPL {X  -147.178, Y  +734.233, Z    +0.000, E1   +46.439, E3 -305553.256}
SPL {X  -140.263, Y  +748.461, Z    +0.000, E1   +42.675, E3 -305611.594}
ENDSPLINE

SPLINE
SPL {X  -141.835, Y  +745.525, Z    +0.000, E1   +39.068, E3 -305643.595}
SPL {X  -152.406, Y  +720.176, Z    +0.000, E1   +27.814, E3 -305694.808}
SPL {X  -157.542, Y  +699.382, Z    +0.000, E1   +18.086, E3 -305709.141}
SPL {X  -159.386, Y  +685.393, Z    +0.000, E1   +10.664, E3 -305714.095}
SPL {X  -159.928, Y  +675.946, Z    +0.000, E1    +5.007, E3 -305716.134}
SPL {X  -159.990, Y  +671.468, Z    +0.000, E1    +2.030, E3 -305716.730}
SPL {X  -159.990, Y  +667.678, Z    +0.000, E1    -0.783, E3 -305717.080}
SPL {X  -159.990, Y  +663.139, Z    +0.000, E1    -5.135, E3 -305717.597}
SPL {X  -159.990, Y  +658.551, Z    +0.000, E1   -10.313, E3 -305718.371}
SPL {X  -159.990, Y  +653.526, Z    +0.000, E1   -16.156, E3 -305719.606}
SPL {X  -159.990, Y  +644.434, Z    +0.000, E1   -25.921, E3 -305722.801}
SPL {X  -159.990, Y  +612.255, Z    +0.000, E1   -44.102, E3 -305744.682}
SPL {X  -159.990, Y  +561.053, Z    +0.000, E1   -49.668, E3 -305809.515}
SPL {X  -159.990, Y  +552.984, Z    +0.000, E1   -49.619, E3 -305824.156}
SPL {X  -159.990, Y  +547.278, Z    +0.000, E1   -49.619, E3 -305834.455}
SPL {X  -159.990, Y  +538.738, Z    +0.000, E1   -49.672, E3 -305849.779}
SPL {X  -159.990, Y  +529.436, Z    +0.000, E1   -49.638, E3 -305866.603}
SPL {X  -159.990, Y  +520.280, Z    +0.000, E1   -49.665, E3 -305883.082}
SPL {X  -159.990, Y  +511.038, Z    +0.000, E1   -49.636, E3 -305899.832}
SPL {X  -159.990, Y  +504.260, Z    +0.000, E1   -49.614, E3 -305912.105}
SPL {X  -159.990, Y  +503.881, Z    +0.000, E1   -48.376, E3 -305920.092}
ENDSPLINE

SPLINE
SPL {X  -159.990, Y  +520.622, Z    +0.000, E1   -41.395, E3 -305926.672}
ENDSPLINE

